LIN {X 0,Y 362.769,Z 567.893,A -85,B 0,C 180,E1 -12881.17,E2 -12881.17} C_VEL
LIN {X 0,Y 361.723,Z 575.209,A -85,B 0,C 180,E1 -12883.722,E2 -12883.722} C_VEL
LIN {X 0,Y 361.091,Z 580.078,A -85,B 0,C 180,E1 -12885.812,E2 -12885.812} C_VEL
LIN {X 0,Y 360.592,Z 584.335,A -85,B 0,C 180,E1 -12888.17,E2 -12888.17} C_VEL
LIN {X 0,Y 360.281,Z 587.529,A -85,B 0,C 180,E1 -12890.556,E2 -12890.556} C_VEL
LIN {X 0,Y 360.062,Z 589.612,A -85,B 0,C 180,E1 -12892.977,E2 -12892.977} C_VEL
LIN {X 0,Y 360.017,Z 590.544,A -85,B 0,C 180,E1 -12895.433,E2 -12895.433} C_VEL
LIN {X 0,Y 360.084,Z 590.365,A -85,B 0,C 180,E1 -12897.931,E2 -12897.931} C_VEL
LIN {X 0,Y 360.211,Z 588.944,A -85,B 0,C 180,E1 -12900.482,E2 -12900.482} C_VEL
LIN {X 0,Y 360.536,Z 586.171,A -85,B 0,C 180,E1 -12903.079,E2 -12903.079} C_VEL
LIN {X 0,Y 361.081,Z 581.98,A -85,B 0,C 180,E1 -12905.725,E2 -12905.725} C_VEL
LIN {X 0,Y 361.82,Z 576.187,A -85,B 0,C 180,E1 -12908.43,E2 -12908.43} C_VEL
LIN {X 0,Y 362.912,Z 569.264,A -85,B 0,C 180,E1 -12910.952,E2 -12910.952} C_VEL
LIN {X 0,Y 364.311,Z 561.304,A -85,B 0,C 180,E1 -12913.307,E2 -12913.307} C_VEL
LIN {X 0,Y 366.113,Z 551.646,A -85,B 0,C 180,E1 -12915.647,E2 -12915.647} C_VEL
LIN {X 0,Y 368.136,Z 541.41,A -85,B 0,C 180,E1 -12917.71,E2 -12917.71} C_VEL
LIN {X 0,Y 370.476,Z 529.462,A -85,B 0,C 180,E1 -12919.738,E2 -12919.738} C_VEL
LIN {X 0,Y 372.823,Z 516.873,A -85,B 0,C 180,E1 -12921.532,E2 -12921.532} C_VEL
LIN {X 0,Y 375.168,Z 504.129,A -85,B 0,C 180,E1 -12923.058,E2 -12923.058} C_VEL
LIN {X 0,Y 377.529,Z 489.396,A -85,B 0,C 180,E1 -12924.53,E2 -12924.53} C_VEL
LIN {X 0,Y 379.798,Z 473.918,A -85,B 0,C 180,E1 -12925.782,E2 -12925.782} C_VEL
LIN {X 0,Y 381.548,Z 459.656,A -85,B 0,C 180,E1 -12926.719,E2 -12926.719} C_VEL
LIN {X 0,Y 383.185,Z 443.468,A -85,B 0,C 180,E1 -12927.561,E2 -12927.561} C_VEL
LIN {X 0,Y 384.533,Z 426.825,A -85,B 0,C 180,E1 -12928.196,E2 -12928.196} C_VEL
LIN {X 0,Y 385.454,Z 409.688,A -85,B 0,C 180,E1 -12928.632,E2 -12928.632} C_VEL
LIN {X 0,Y 390.375,Z 262.96,A -85,B 0,C 180,E1 -12931.532,E2 -12931.532} C_VEL
LIN {X 0,Y 381.789,Z 246.096,A -85,B 0,C 180,E1 -12932.964,E2 -12932.964} C_VEL
LIN {X 0,Y 375.213,Z 234.438,A -85,B 0,C 180,E1 -12934.104,E2 -12934.104} C_VEL
LIN {X 0,Y 367.237,Z 221.553,A -85,B 0,C 180,E1 -12935.553,E2 -12935.553} C_VEL
LIN {X 0,Y 365.03,Z 218.312,A -85,B 0,C 180,E1 -12935.963,E2 -12935.963} C_VEL
LIN {X 0,Y 362.546,Z 214.885,A -85,B 0,C 180,E1 -12936.433,E2 -12936.433} C_VEL
LIN {X 0,Y 362.042,Z 213.576,A -85,B 0,C 180,E1 -12936.55,E2 -12936.55} C_VEL
LIN {X 0,Y 361.879,Z 212.722,A -85,B 0,C 180,E1 -12936.766,E2 -12936.766} C_VEL
LIN {X 0,Y 361.879,Z 212.713,A -85,B 0,C 180,E1 -12940.722,E2 -12940.722} C_VEL
LIN {X 0,Y 361.937,Z 212.702,A -85,B 0,C 180,E1 -12944.226,E2 -12944.226} C_VEL
LIN {X 0,Y 361.993,Z 212.706,A -85,B 0,C 180,E1 -12946.528,E2 -12946.528} C_VEL
LIN {X 0,Y 361.994,Z 212.706,A -85,B 0,C 180,E1 -12949.937,E2 -12949.937} C_VEL
LIN {X 0,Y 362.142,Z 212.683,A -85,B 0,C 180,E1 -12953.313,E2 -12953.313} C_VEL
LIN {X 0,Y 362.274,Z 212.669,A -85,B 0,C 180,E1 -12957.776,E2 -12957.776} C_VEL
LIN {X 0,Y 362.421,Z 212.652,A -85,B 0,C 180,E1 -12960,E2 -12960} C_VEL
LIN {X 0,Y 362.274,Z 212.671,A -85,B 0,C 180,E1 -12962.224,E2 -12962.224} C_VEL
LIN {X 0,Y 362.157,Z 212.687,A -85,B 0,C 180,E1 -12966.686,E2 -12966.686} C_VEL
LIN {X 0,Y 362.025,Z 212.703,A -85,B 0,C 180,E1 -12970.062,E2 -12970.062} C_VEL
LIN {X 0,Y 361.992,Z 212.703,A -85,B 0,C 180,E1 -12973.899,E2 -12973.899} C_VEL
LIN {X 0,Y 361.962,Z 212.711,A -85,B 0,C 180,E1 -12977.939,E2 -12977.939} C_VEL
LIN {X 0,Y 361.886,Z 212.717,A -85,B 0,C 180,E1 -12981.653,E2 -12981.653} C_VEL
LIN {X 0,Y 361.923,Z 212.715,A -85,B 0,C 180,E1 -12985.29,E2 -12985.29} C_VEL
LIN {X 0,Y 361.903,Z 212.721,A -85,B 0,C 180,E1 -12987.779,E2 -12987.779} C_VEL
LIN {X 0,Y 361.832,Z 212.726,A -85,B 0,C 180,E1 -12991.63,E2 -12991.63} C_VEL
LIN {X 0,Y 361.869,Z 212.725,A -85,B 0,C 180,E1 -12995.345,E2 -12995.345} C_VEL
LIN {X 0,Y 361.865,Z 212.73,A -85,B 0,C 180,E1 -12999.027,E2 -12999.027} C_VEL
LIN {X 0,Y 361.831,Z 212.734,A -85,B 0,C 180,E1 -13002.829,E2 -13002.829} C_VEL
LIN {X 0,Y 361.843,Z 212.773,A -85,B 0,C 180,E1 -13006.82,E2 -13006.82} C_VEL
LIN {X 0,Y 367.527,Z 227.558,A -85,B 0,C 180,E1 -13010.269,E2 -13010.269} C_VEL
LIN {X 0,Y 376.278,Z 242.828,A -85,B 0,C 180,E1 -13011.891,E2 -13011.891} C_VEL
LIN {X 0,Y 384.124,Z 257.902,A -85,B 0,C 180,E1 -13013.252,E2 -13013.252} C_VEL
LIN {X 0,Y 389.455,Z 269.218,A -85,B 0,C 180,E1 -13014.151,E2 -13014.151} C_VEL
LIN {X 0,Y 390.123,Z 274.919,A -85,B 0,C 180,E1 -13014.361,E2 -13014.361} C_VEL
LIN {X 0,Y 384.621,Z 436.732,A -85,B 0,C 180,E1 -13017.579,E2 -13017.579} C_VEL
LIN {X 0,Y 383.351,Z 452.919,A -85,B 0,C 180,E1 -13018.077,E2 -13018.077} C_VEL
LIN {X 0,Y 381.853,Z 468.395,A -85,B 0,C 180,E1 -13018.75,E2 -13018.75} C_VEL
LIN {X 0,Y 380.022,Z 483.398,A -85,B 0,C 180,E1 -13019.586,E2 -13019.586} C_VEL
LIN {X 0,Y 377.904,Z 498.273,A -85,B 0,C 180,E1 -13020.627,E2 -13020.627} C_VEL
LIN {X 0,Y 375.599,Z 513.155,A -85,B 0,C 180,E1 -13021.923,E2 -13021.923} C_VEL
LIN {X 0,Y 373.038,Z 527.462,A -85,B 0,C 180,E1 -13023.421,E2 -13023.421} C_VEL
LIN {X 0,Y 370.694,Z 540.406,A -85,B 0,C 180,E1 -13025.05,E2 -13025.05} C_VEL
LIN {X 0,Y 368.649,Z 551.565,A -85,B 0,C 180,E1 -13026.698,E2 -13026.698} C_VEL
LIN {X 0,Y 366.587,Z 562.673,A -85,B 0,C 180,E1 -13028.639,E2 -13028.639} C_VEL
LIN {X 0,Y 364.623,Z 573.214,A -85,B 0,C 180,E1 -13030.814,E2 -13030.814} C_VEL
LIN {X 0,Y 363.105,Z 582.549,A -85,B 0,C 180,E1 -13033.123,E2 -13033.123} C_VEL
LIN {X 0,Y 361.954,Z 590.186,A -85,B 0,C 180,E1 -13035.38,E2 -13035.38} C_VEL
LIN {X 0,Y 361.04,Z 597.839,A -85,B 0,C 180,E1 -13038.207,E2 -13038.207} C_VEL
LIN {X 0,Y 360.52,Z 603.683,A -85,B 0,C 180,E1 -13041.028,E2 -13041.028} C_VEL
LIN {X 0,Y 360.379,Z 607.096,A -85,B 0,C 180,E1 -13043.281,E2 -13043.281} C_VEL
LIN {X 0,Y 360.298,Z 609.553,A -85,B 0,C 180,E1 -13045.525,E2 -13045.525} C_VEL
LIN {X 0,Y 360.27,Z 610.947,A -85,B 0,C 180,E1 -13047.764,E2 -13047.764} C_VEL
LIN {X 0,Y 360.356,Z 611.428,A -85,B 0,C 180,E1 -13050,E2 -13050} C_VEL
LIN {X 0,Y 360.272,Z 610.861,A -85,B 0,C 180,E1 -13052.236,E2 -13052.236} C_VEL
LIN {X 0,Y 360.298,Z 609.372,A -85,B 0,C 180,E1 -13054.475,E2 -13054.475} C_VEL
LIN {X 0,Y 360.379,Z 606.819,A -85,B 0,C 180,E1 -13056.72,E2 -13056.72} C_VEL
LIN {X 0,Y 360.521,Z 603.263,A -85,B 0,C 180,E1 -13058.972,E2 -13058.972} C_VEL
LIN {X 0,Y 360.875,Z 598.584,A -85,B 0,C 180,E1 -13061.23,E2 -13061.23} C_VEL
LIN {X 0,Y 361.623,Z 592.232,A -85,B 0,C 180,E1 -13063.657,E2 -13063.657} C_VEL
LIN {X 0,Y 362.564,Z 584.596,A -85,B 0,C 180,E1 -13066.035,E2 -13066.035} C_VEL
LIN {X 0,Y 363.903,Z 575.912,A -85,B 0,C 180,E1 -13068.277,E2 -13068.277} C_VEL
LIN {X 0,Y 365.602,Z 565.37,A -85,B 0,C 180,E1 -13070.538,E2 -13070.538} C_VEL
LIN {X 0,Y 367.5,Z 554.478,A -85,B 0,C 180,E1 -13072.487,E2 -13072.487} C_VEL
LIN {X 0,Y 369.418,Z 543.389,A -85,B 0,C 180,E1 -13074.185,E2 -13074.185} C_VEL
LIN {X 0,Y 371.553,Z 531.128,A -85,B 0,C 180,E1 -13075.788,E2 -13075.788} C_VEL
LIN {X 0,Y 373.767,Z 517.501,A -85,B 0,C 180,E1 -13077.279,E2 -13077.279} C_VEL
LIN {X 0,Y 375.967,Z 503.055,A -85,B 0,C 180,E1 -13078.591,E2 -13078.591} C_VEL
LIN {X 0,Y 377.997,Z 488.557,A -85,B 0,C 180,E1 -13079.672,E2 -13079.672} C_VEL
LIN {X 0,Y 379.777,Z 473.42,A -85,B 0,C 180,E1 -13080.591,E2 -13080.591} C_VEL
LIN {X 0,Y 381.381,Z 455.748,A -85,B 0,C 180,E1 -13081.41,E2 -13081.41} C_VEL
LIN {X 0,Y 382.692,Z 438.69,A -85,B 0,C 180,E1 -13081.947,E2 -13081.947} C_VEL
LIN {X 0,Y 383.543,Z 416.513,A -85,B 0,C 180,E1 -13082.407,E2 -13082.407} C_VEL
LIN {X 0,Y 387.858,Z 273.203,A -85,B 0,C 180,E1 -13085.197,E2 -13085.197} C_VEL
LIN {X 0,Y 386.788,Z 267.489,A -85,B 0,C 180,E1 -13085.431,E2 -13085.431} C_VEL
LIN {X 0,Y 376.132,Z 245.181,A -85,B 0,C 180,E1 -13087.042,E2 -13087.042} C_VEL
LIN {X 0,Y 367.589,Z 229.114,A -85,B 0,C 180,E1 -13088.383,E2 -13088.383} C_VEL
LIN {X 0,Y 362.976,Z 216.179,A -85,B 0,C 180,E1 -13090.964,E2 -13090.964} C_VEL
LIN {X 0,Y 361.842,Z 212.725,A -85,B 0,C 180,E1 -13091.692,E2 -13091.692} C_VEL
LIN {X 0,Y 361.814,Z 212.718,A -85,B 0,C 180,E1 -13095.631,E2 -13095.631} C_VEL
LIN {X 0,Y 361.827,Z 212.716,A -85,B 0,C 180,E1 -13099.246,E2 -13099.246} C_VEL
LIN {X 0,Y 361.863,Z 212.71,A -85,B 0,C 180,E1 -13102.982,E2 -13102.982} C_VEL
LIN {X 0,Y 361.856,Z 212.721,A -85,B 0,C 180,E1 -13106.631,E2 -13106.631} C_VEL
LIN {X 0,Y 361.871,Z 212.714,A -85,B 0,C 180,E1 -13109.672,E2 -13109.672} C_VEL
LIN {X 0,Y 361.951,Z 212.692,A -85,B 0,C 180,E1 -13113.475,E2 -13113.475} C_VEL
LIN {X 0,Y 361.888,Z 212.721,A -85,B 0,C 180,E1 -13117.145,E2 -13117.145} C_VEL
LIN {X 0,Y 361.883,Z 212.693,A -85,B 0,C 180,E1 -13120.722,E2 -13120.722} C_VEL
LIN {X 0,Y 361.941,Z 212.713,A -85,B 0,C 180,E1 -13124.226,E2 -13124.226} C_VEL
LIN {X 0,Y 361.996,Z 212.689,A -85,B 0,C 180,E1 -13126.528,E2 -13126.528} C_VEL
LIN {X 0,Y 361.997,Z 212.686,A -85,B 0,C 180,E1 -13129.937,E2 -13129.937} C_VEL
LIN {X 0,Y 362.146,Z 212.684,A -85,B 0,C 180,E1 -13133.313,E2 -13133.313} C_VEL
LIN {X 0,Y 362.277,Z 212.634,A -85,B 0,C 180,E1 -13137.776,E2 -13137.776} C_VEL
LIN {X 0,Y 362.423,Z 212.643,A -85,B 0,C 180,E1 -13140,E2 -13140} C_VEL
LIN {X 0,Y 362.277,Z 212.671,A -85,B 0,C 180,E1 -13142.224,E2 -13142.224} C_VEL
LIN {X 0,Y 362.16,Z 212.678,A -85,B 0,C 180,E1 -13146.686,E2 -13146.686} C_VEL
LIN {X 0,Y 362.028,Z 212.694,A -85,B 0,C 180,E1 -13150.062,E2 -13150.062} C_VEL
LIN {X 0,Y 361.996,Z 212.697,A -85,B 0,C 180,E1 -13153.899,E2 -13153.899} C_VEL
LIN {X 0,Y 361.965,Z 212.691,A -85,B 0,C 180,E1 -13157.939,E2 -13157.939} C_VEL
LIN {X 0,Y 361.89,Z 212.717,A -85,B 0,C 180,E1 -13161.653,E2 -13161.653} C_VEL
LIN {X 0,Y 361.926,Z 212.696,A -85,B 0,C 180,E1 -13165.29,E2 -13165.29} C_VEL
LIN {X 0,Y 361.921,Z 212.712,A -85,B 0,C 180,E1 -13167.778,E2 -13167.778} C_VEL
LIN {X 0,Y 361.845,Z 212.711,A -85,B 0,C 180,E1 -13171.285,E2 -13171.285} C_VEL
LIN {X 0,Y 361.853,Z 212.723,A -85,B 0,C 180,E1 -13174.28,E2 -13174.28} C_VEL
LIN {X 0,Y 361.863,Z 212.712,A -85,B 0,C 180,E1 -13177.223,E2 -13177.223} C_VEL
LIN {X 0,Y 361.835,Z 212.724,A -85,B 0,C 180,E1 -13180.756,E2 -13180.756} C_VEL
LIN {X 0,Y 361.815,Z 212.717,A -85,B 0,C 180,E1 -13184.369,E2 -13184.369} C_VEL
LIN {X 0,Y 361.834,Z 212.721,A -85,B 0,C 180,E1 -13187.568,E2 -13187.568} C_VEL
LIN {X 0,Y 361.867,Z 212.72,A -85,B 0,C 180,E1 -13190.974,E2 -13190.974} C_VEL
LIN {X 0,Y 361.873,Z 212.71,A -85,B 0,C 180,E1 -13194.655,E2 -13194.655} C_VEL
LIN {X 0,Y 361.836,Z 212.714,A -85,B 0,C 180,E1 -13198.371,E2 -13198.371} C_VEL
LIN {X 0,Y 361.9,Z 212.721,A -85,B 0,C 180,E1 -13200.955,E2 -13200.955} C_VEL
LIN {X 0,Y 361.953,Z 212.705,A -85,B 0,C 180,E1 -13203.475,E2 -13203.475} C_VEL
LIN {X 0,Y 361.892,Z 212.714,A -85,B 0,C 180,E1 -13207.145,E2 -13207.145} C_VEL
LIN {X 0,Y 361.887,Z 212.689,A -85,B 0,C 180,E1 -13210.722,E2 -13210.722} C_VEL
LIN {X 0,Y 361.933,Z 212.711,A -85,B 0,C 180,E1 -13213.066,E2 -13213.066} C_VEL
LIN {X 0,Y 362.024,Z 212.683,A -85,B 0,C 180,E1 -13217.039,E2 -13217.039} C_VEL
LIN {X 0,Y 363.054,Z 215.611,A -85,B 0,C 180,E1 -13217.248,E2 -13217.248} C_VEL
LIN {X 0,Y 364.548,Z 217.745,A -85,B 0,C 180,E1 -13217.479,E2 -13217.479} C_VEL
LIN {X 0,Y 373.522,Z 232.837,A -85,B 0,C 180,E1 -13218.87,E2 -13218.87} C_VEL
LIN {X 0,Y 381.962,Z 248.896,A -85,B 0,C 180,E1 -13220.142,E2 -13220.142} C_VEL
LIN {X 0,Y 388.027,Z 261.925,A -85,B 0,C 180,E1 -13221.052,E2 -13221.052} C_VEL
LIN {X 0,Y 383.18,Z 416.866,A -85,B 0,C 180,E1 -13224.078,E2 -13224.078} C_VEL
LIN {X 0,Y 382.141,Z 433.477,A -85,B 0,C 180,E1 -13224.591,E2 -13224.591} C_VEL
LIN {X 0,Y 380.8,Z 449.353,A -85,B 0,C 180,E1 -13225.284,E2 -13225.284} C_VEL
LIN {X 0,Y 379.228,Z 464.561,A -85,B 0,C 180,E1 -13226.148,E2 -13226.148} C_VEL
LIN {X 0,Y 377.475,Z 479.265,A -85,B 0,C 180,E1 -13227.198,E2 -13227.198} C_VEL
LIN {X 0,Y 375.491,Z 493,A -85,B 0,C 180,E1 -13228.391,E2 -13228.391} C_VEL
LIN {X 0,Y 373.256,Z 507.153,A -85,B 0,C 180,E1 -13229.865,E2 -13229.865} C_VEL
LIN {X 0,Y 371.296,Z 519.204,A -85,B 0,C 180,E1 -13231.355,E2 -13231.355} C_VEL
LIN {X 0,Y 368.932,Z 532.288,A -85,B 0,C 180,E1 -13233.276,E2 -13233.276} C_VEL
LIN {X 0,Y 366.965,Z 543.218,A -85,B 0,C 180,E1 -13235.201,E2 -13235.201} C_VEL
LIN {X 0,Y 365.295,Z 552.773,A -85,B 0,C 180,E1 -13237.184,E2 -13237.184} C_VEL
LIN {X 0,Y 364.07,Z 559.988,A -85,B 0,C 180,E1 -13238.919,E2 -13238.919} C_VEL
LIN {X 0,Y 362.924,Z 563.011,A -85,B 0,C 180,E1 -13239.699,E2 -13239.699} C_VEL
LIN {X 0,Y 356.43,Z 571.259,A -85,B 0,C 180,E1 -13242.006,E2 -13242.006} C_VEL
LIN {X 0,Y 355.052,Z 573.747,A -85,B 0,C 180,E1 -13242.844,E2 -13242.844} C_VEL
LIN {X 0,Y 354.865,Z 574.488,A -85,B 0,C 180,E1 -13243.134,E2 -13243.134} C_VEL
LIN {X 0,Y 354.076,Z 580.085,A -85,B 0,C 180,E1 -13245.542,E2 -13245.542} C_VEL
LIN {X 0,Y 353.644,Z 583.644,A -85,B 0,C 180,E1 -13247.464,E2 -13247.464} C_VEL
LIN {X 0,Y 353.257,Z 586.927,A -85,B 0,C 180,E1 -13249.767,E2 -13249.767} C_VEL
LIN {X 0,Y 352.994,Z 589.314,A -85,B 0,C 180,E1 -13252.227,E2 -13252.227} C_VEL
LIN {X 0,Y 352.916,Z 590.638,A -85,B 0,C 180,E1 -13254.72,E2 -13254.72} C_VEL
LIN {X 0,Y 352.949,Z 590.735,A -85,B 0,C 180,E1 -13257.256,E2 -13257.256} C_VEL
LIN {X 0,Y 353.05,Z 589.663,A -85,B 0,C 180,E1 -13259.845,E2 -13259.845} C_VEL
LIN {X 0,Y 353.334,Z 587.334,A -85,B 0,C 180,E1 -13262.482,E2 -13262.482} C_VEL
LIN {X 0,Y 353.885,Z 583.591,A -85,B 0,C 180,E1 -13265.164,E2 -13265.164} C_VEL
LIN {X 0,Y 354.582,Z 578.249,A -85,B 0,C 180,E1 -13267.91,E2 -13267.91} C_VEL
LIN {X 0,Y 355.418,Z 572.986,A -85,B 0,C 180,E1 -13270.04,E2 -13270.04} C_VEL
LIN {X 0,Y 356.46,Z 566.926,A -85,B 0,C 180,E1 -13272.093,E2 -13272.093} C_VEL
LIN {X 0,Y 358.153,Z 558.136,A -85,B 0,C 180,E1 -13274.548,E2 -13274.548} C_VEL
LIN {X 0,Y 359.902,Z 549.284,A -85,B 0,C 180,E1 -13276.618,E2 -13276.618} C_VEL
LIN {X 0,Y 362.163,Z 538.628,A -85,B 0,C 180,E1 -13278.716,E2 -13278.716} C_VEL
LIN {X 0,Y 364.59,Z 526.833,A -85,B 0,C 180,E1 -13280.665,E2 -13280.665} C_VEL
LIN {X 0,Y 366.84,Z 514.974,A -85,B 0,C 180,E1 -13282.316,E2 -13282.316} C_VEL
LIN {X 0,Y 369.3,Z 501.917,A -85,B 0,C 180,E1 -13283.847,E2 -13283.847} C_VEL
LIN {X 0,Y 371.611,Z 488.087,A -85,B 0,C 180,E1 -13285.213,E2 -13285.213} C_VEL
LIN {X 0,Y 373.844,Z 473.322,A -85,B 0,C 180,E1 -13286.411,E2 -13286.411} C_VEL
LIN {X 0,Y 375.816,Z 457.752,A -85,B 0,C 180,E1 -13287.424,E2 -13287.424} C_VEL
LIN {X 0,Y 377.404,Z 441.921,A -85,B 0,C 180,E1 -13288.233,E2 -13288.233} C_VEL
LIN {X 0,Y 378.794,Z 425.309,A -85,B 0,C 180,E1 -13288.845,E2 -13288.845} C_VEL
LIN {X 0,Y 379.651,Z 408.154,A -85,B 0,C 180,E1 -13289.274,E2 -13289.274} C_VEL
LIN {X 0,Y 384.65,Z 265.3,A -85,B 0,C 180,E1 -13292.141,E2 -13292.141} C_VEL
LIN {X 0,Y 377.068,Z 250.316,A -85,B 0,C 180,E1 -13293.451,E2 -13293.451} C_VEL
LIN {X 0,Y 369.948,Z 237.666,A -85,B 0,C 180,E1 -13294.733,E2 -13294.733} C_VEL
LIN {X 0,Y 363.101,Z 226.601,A -85,B 0,C 180,E1 -13296.017,E2 -13296.017} C_VEL
LIN {X 0,Y 359.879,Z 221.971,A -85,B 0,C 180,E1 -13296.639,E2 -13296.639} C_VEL
LIN {X 0,Y 357.501,Z 218.319,A -85,B 0,C 180,E1 -13297.116,E2 -13297.116} C_VEL
LIN {X 0,Y 355.465,Z 215.85,A -85,B 0,C 180,E1 -13297.515,E2 -13297.515} C_VEL
LIN {X 0,Y 354.797,Z 213.63,A -85,B 0,C 180,E1 -13297.738,E2 -13297.738} C_VEL
LIN {X 0,Y 354.841,Z 213.591,A -85,B 0,C 180,E1 -13301.525,E2 -13301.525} C_VEL
LIN {X 0,Y 354.913,Z 213.58,A -85,B 0,C 180,E1 -13305.083,E2 -13305.083} C_VEL
LIN {X 0,Y 354.927,Z 213.573,A -85,B 0,C 180,E1 -13308.579,E2 -13308.579} C_VEL
LIN {X 0,Y 355.055,Z 213.57,A -85,B 0,C 180,E1 -13312.036,E2 -13312.036} C_VEL
LIN {X 0,Y 355.077,Z 213.568,A -85,B 0,C 180,E1 -13314.32,E2 -13314.32} C_VEL
LIN {X 0,Y 355.237,Z 213.546,A -85,B 0,C 180,E1 -13317.732,E2 -13317.732} C_VEL
LIN {X 0,Y 355.391,Z 213.528,A -85,B 0,C 180,E1 -13320,E2 -13320} C_VEL
LIN {X 0,Y 355.237,Z 213.547,A -85,B 0,C 180,E1 -13322.268,E2 -13322.268} C_VEL
LIN {X 0,Y 355.12,Z 213.563,A -85,B 0,C 180,E1 -13326.82,E2 -13326.82} C_VEL
LIN {X 0,Y 354.972,Z 213.579,A -85,B 0,C 180,E1 -13330.264,E2 -13330.264} C_VEL
LIN {X 0,Y 354.937,Z 213.582,A -85,B 0,C 180,E1 -13334.019,E2 -13334.019} C_VEL
LIN {X 0,Y 354.917,Z 213.587,A -85,B 0,C 180,E1 -13338.109,E2 -13338.109} C_VEL
LIN {X 0,Y 354.829,Z 213.596,A -85,B 0,C 180,E1 -13342.106,E2 -13342.106} C_VEL
LIN {X 0,Y 354.894,Z 213.59,A -85,B 0,C 180,E1 -13345.828,E2 -13345.828} C_VEL
LIN {X 0,Y 354.812,Z 213.6,A -85,B 0,C 180,E1 -13349.682,E2 -13349.682} C_VEL
LIN {X 0,Y 354.801,Z 213.603,A -85,B 0,C 180,E1 -13353.702,E2 -13353.702} C_VEL
LIN {X 0,Y 354.793,Z 213.607,A -85,B 0,C 180,E1 -13356.46,E2 -13356.46} C_VEL
LIN {X 0,Y 354.819,Z 213.606,A -85,B 0,C 180,E1 -13359.424,E2 -13359.424} C_VEL
LIN {X 0,Y 354.783,Z 213.613,A -85,B 0,C 180,E1 -13362.868,E2 -13362.868} C_VEL
LIN {X 0,Y 354.792,Z 213.641,A -85,B 0,C 180,E1 -13365.814,E2 -13365.814} C_VEL
LIN {X 0,Y 360.125,Z 227.357,A -85,B 0,C 180,E1 -13369.185,E2 -13369.185} C_VEL
LIN {X 0,Y 367.513,Z 239.811,A -85,B 0,C 180,E1 -13370.623,E2 -13370.623} C_VEL
LIN {X 0,Y 375.875,Z 255.03,A -85,B 0,C 180,E1 -13372.154,E2 -13372.154} C_VEL
LIN {X 0,Y 384.139,Z 272.385,A -85,B 0,C 180,E1 -13373.61,E2 -13373.61} C_VEL
LIN {X 0,Y 384.462,Z 276.603,A -85,B 0,C 180,E1 -13373.751,E2 -13373.751} C_VEL
LIN {X 0,Y 378.761,Z 436.245,A -85,B 0,C 180,E1 -13376.966,E2 -13376.966} C_VEL
LIN {X 0,Y 377.442,Z 452.666,A -85,B 0,C 180,E1 -13377.477,E2 -13377.477} C_VEL
LIN {X 0,Y 375.956,Z 467.472,A -85,B 0,C 180,E1 -13378.124,E2 -13378.124} C_VEL
LIN {X 0,Y 374.219,Z 481.6,A -85,B 0,C 180,E1 -13378.906,E2 -13378.906} C_VEL
LIN {X 0,Y 371.996,Z 496.641,A -85,B 0,C 180,E1 -13379.957,E2 -13379.957} C_VEL
LIN {X 0,Y 369.786,Z 510.587,A -85,B 0,C 180,E1 -13381.155,E2 -13381.155} C_VEL
LIN {X 0,Y 367.362,Z 523.948,A -85,B 0,C 180,E1 -13382.515,E2 -13382.515} C_VEL
LIN {X 0,Y 364.801,Z 537.406,A -85,B 0,C 180,E1 -13384.16,E2 -13384.16} C_VEL
LIN {X 0,Y 362.4,Z 549.736,A -85,B 0,C 180,E1 -13385.968,E2 -13385.968} C_VEL
LIN {X 0,Y 360.152,Z 561.093,A -85,B 0,C 180,E1 -13387.937,E2 -13387.937} C_VEL
LIN {X 0,Y 358.026,Z 572.104,A -85,B 0,C 180,E1 -13390.208,E2 -13390.208} C_VEL
LIN {X 0,Y 356.435,Z 581.396,A -85,B 0,C 180,E1 -13392.501,E2 -13392.501} C_VEL
LIN {X 0,Y 354.994,Z 590.041,A -85,B 0,C 180,E1 -13395.087,E2 -13395.087} C_VEL
LIN {X 0,Y 354.162,Z 596.272,A -85,B 0,C 180,E1 -13397.392,E2 -13397.392} C_VEL
LIN {X 0,Y 353.567,Z 601.354,A -85,B 0,C 180,E1 -13399.695,E2 -13399.695} C_VEL
LIN {X 0,Y 353.358,Z 605.344,A -85,B 0,C 180,E1 -13401.997,E2 -13401.997} C_VEL
LIN {X 0,Y 353.239,Z 608.251,A -85,B 0,C 180,E1 -13404.291,E2 -13404.291} C_VEL
LIN {X 0,Y 353.191,Z 610.189,A -85,B 0,C 180,E1 -13406.578,E2 -13406.578} C_VEL
LIN {X 0,Y 353.218,Z 611.093,A -85,B 0,C 180,E1 -13408.86,E2 -13408.86} C_VEL
LIN {X 0,Y 353.219,Z 611.068,A -85,B 0,C 180,E1 -13411.14,E2 -13411.14} C_VEL
LIN {X 0,Y 353.191,Z 610.008,A -85,B 0,C 180,E1 -13413.423,E2 -13413.423} C_VEL
LIN {X 0,Y 353.275,Z 607.799,A -85,B 0,C 180,E1 -13415.908,E2 -13415.908} C_VEL
LIN {X 0,Y 353.359,Z 604.923,A -85,B 0,C 180,E1 -13418.003,E2 -13418.003} C_VEL
LIN {X 0,Y 353.556,Z 600.84,A -85,B 0,C 180,E1 -13420.306,E2 -13420.306} C_VEL
LIN {X 0,Y 354.369,Z 594.074,A -85,B 0,C 180,E1 -13423.184,E2 -13423.184} C_VEL
LIN {X 0,Y 355.196,Z 587.202,A -85,B 0,C 180,E1 -13425.493,E2 -13425.493} C_VEL
LIN {X 0,Y 356.527,Z 578.965,A -85,B 0,C 180,E1 -13427.791,E2 -13427.791} C_VEL
LIN {X 0,Y 357.876,Z 570.499,A -85,B 0,C 180,E1 -13429.801,E2 -13429.801} C_VEL
LIN {X 0,Y 359.666,Z 560.51,A -85,B 0,C 180,E1 -13431.794,E2 -13431.794} C_VEL
LIN {X 0,Y 361.831,Z 548.841,A -85,B 0,C 180,E1 -13433.768,E2 -13433.768} C_VEL
LIN {X 0,Y 364.076,Z 536.102,A -85,B 0,C 180,E1 -13435.589,E2 -13435.589} C_VEL
LIN {X 0,Y 366.299,Z 523.51,A -85,B 0,C 180,E1 -13437.109,E2 -13437.109} C_VEL
LIN {X 0,Y 368.698,Z 508.886,A -85,B 0,C 180,E1 -13438.57,E2 -13438.57} C_VEL
LIN {X 0,Y 371.003,Z 493.57,A -85,B 0,C 180,E1 -13439.819,E2 -13439.819} C_VEL
LIN {X 0,Y 372.966,Z 478.411,A -85,B 0,C 180,E1 -13440.818,E2 -13440.818} C_VEL
LIN {X 0,Y 374.63,Z 462.494,A -85,B 0,C 180,E1 -13441.647,E2 -13441.647} C_VEL
LIN {X 0,Y 375.968,Z 447.412,A -85,B 0,C 180,E1 -13442.231,E2 -13442.231} C_VEL
LIN {X 0,Y 377.001,Z 431.543,A -85,B 0,C 180,E1 -13442.646,E2 -13442.646} C_VEL
LIN {X 0,Y 381.929,Z 274.277,A -85,B 0,C 180,E1 -13445.762,E2 -13445.762} C_VEL
LIN {X 0,Y 380.971,Z 269.911,A -85,B 0,C 180,E1 -13445.959,E2 -13445.959} C_VEL
LIN {X 0,Y 370.041,Z 247.21,A -85,B 0,C 180,E1 -13447.657,E2 -13447.657} C_VEL
LIN {X 0,Y 360.223,Z 228.821,A -85,B 0,C 180,E1 -13449.258,E2 -13449.258} C_VEL
LIN {X 0,Y 354.812,Z 213.593,A -85,B 0,C 180,E1 -13452.433,E2 -13452.433} C_VEL
LIN {X 0,Y 354.764,Z 213.596,A -85,B 0,C 180,E1 -13456.103,E2 -13456.103} C_VEL
LIN {X 0,Y 354.779,Z 213.594,A -85,B 0,C 180,E1 -13459.178,E2 -13459.178} C_VEL
LIN {X 0,Y 354.799,Z 213.597,A -85,B 0,C 180,E1 -13462.404,E2 -13462.404} C_VEL
LIN {X 0,Y 354.81,Z 213.595,A -85,B 0,C 180,E1 -13464.941,E2 -13464.941} C_VEL
LIN {X 0,Y 354.791,Z 213.585,A -85,B 0,C 180,E1 -13468.405,E2 -13468.405} C_VEL
LIN {X 0,Y 354.844,Z 213.596,A -85,B 0,C 180,E1 -13471.619,E2 -13471.619} C_VEL
LIN {X 0,Y 354.897,Z 213.567,A -85,B 0,C 180,E1 -13474.173,E2 -13474.173} C_VEL
LIN {X 0,Y 354.832,Z 213.598,A -85,B 0,C 180,E1 -13477.894,E2 -13477.894} C_VEL
LIN {X 0,Y 354.887,Z 213.573,A -85,B 0,C 180,E1 -13481.908,E2 -13481.908} C_VEL
LIN {X 0,Y 354.941,Z 213.576,A -85,B 0,C 180,E1 -13485.981,E2 -13485.981} C_VEL
LIN {X 0,Y 354.953,Z 213.562,A -85,B 0,C 180,E1 -13489.735,E2 -13489.735} C_VEL
LIN {X 0,Y 355.109,Z 213.561,A -85,B 0,C 180,E1 -13493.18,E2 -13493.18} C_VEL
LIN {X 0,Y 355.24,Z 213.509,A -85,B 0,C 180,E1 -13497.732,E2 -13497.732} C_VEL
LIN {X 0,Y 355.372,Z 213.521,A -85,B 0,C 180,E1 -13500,E2 -13500} C_VEL
LIN {X 0,Y 355.241,Z 213.547,A -85,B 0,C 180,E1 -13502.268,E2 -13502.268} C_VEL
LIN {X 0,Y 355.124,Z 213.556,A -85,B 0,C 180,E1 -13506.819,E2 -13506.819} C_VEL
LIN {X 0,Y 354.975,Z 213.569,A -85,B 0,C 180,E1 -13510.264,E2 -13510.264} C_VEL
LIN {X 0,Y 354.941,Z 213.577,A -85,B 0,C 180,E1 -13514.019,E2 -13514.019} C_VEL
LIN {X 0,Y 354.92,Z 213.566,A -85,B 0,C 180,E1 -13518.108,E2 -13518.108} C_VEL
LIN {X 0,Y 354.833,Z 213.599,A -85,B 0,C 180,E1 -13522.106,E2 -13522.106} C_VEL
LIN {X 0,Y 354.897,Z 213.571,A -85,B 0,C 180,E1 -13525.827,E2 -13525.827} C_VEL
LIN {X 0,Y 354.853,Z 213.594,A -85,B 0,C 180,E1 -13529.679,E2 -13529.679} C_VEL
LIN {X 0,Y 354.804,Z 213.594,A -85,B 0,C 180,E1 -13533.702,E2 -13533.702} C_VEL
LIN {X 0,Y 354.797,Z 213.597,A -85,B 0,C 180,E1 -13536.459,E2 -13536.459} C_VEL
LIN {X 0,Y 354.823,Z 213.589,A -85,B 0,C 180,E1 -13539.424,E2 -13539.424} C_VEL
LIN {X 0,Y 354.786,Z 213.596,A -85,B 0,C 180,E1 -13542.867,E2 -13542.867} C_VEL
LIN {X 0,Y 354.766,Z 213.606,A -85,B 0,C 180,E1 -13546.104,E2 -13546.104} C_VEL
LIN {X 0,Y 354.785,Z 213.591,A -85,B 0,C 180,E1 -13549.179,E2 -13549.179} C_VEL
LIN {X 0,Y 354.805,Z 213.598,A -85,B 0,C 180,E1 -13552.403,E2 -13552.403} C_VEL
LIN {X 0,Y 354.81,Z 213.591,A -85,B 0,C 180,E1 -13554.941,E2 -13554.941} C_VEL
LIN {X 0,Y 354.792,Z 213.591,A -85,B 0,C 180,E1 -13558.405,E2 -13558.405} C_VEL
LIN {X 0,Y 354.848,Z 213.592,A -85,B 0,C 180,E1 -13561.619,E2 -13561.619} C_VEL
LIN {X 0,Y 354.899,Z 213.589,A -85,B 0,C 180,E1 -13564.173,E2 -13564.173} C_VEL
LIN {X 0,Y 354.836,Z 213.599,A -85,B 0,C 180,E1 -13567.894,E2 -13567.894} C_VEL
LIN {X 0,Y 354.922,Z 213.561,A -85,B 0,C 180,E1 -13571.892,E2 -13571.892} C_VEL
LIN {X 0,Y 354.942,Z 213.559,A -85,B 0,C 180,E1 -13575.981,E2 -13575.981} C_VEL
LIN {X 0,Y 354.952,Z 213.562,A -85,B 0,C 180,E1 -13576.212,E2 -13576.212} C_VEL
LIN {X 0,Y 355.962,Z 216.419,A -85,B 0,C 180,E1 -13576.412,E2 -13576.412} C_VEL
LIN {X 0,Y 357.581,Z 218.616,A -85,B 0,C 180,E1 -13576.668,E2 -13576.668} C_VEL
LIN {X 0,Y 368.368,Z 236.593,A -85,B 0,C 180,E1 -13578.388,E2 -13578.388} C_VEL
LIN {X 0,Y 376.777,Z 252.688,A -85,B 0,C 180,E1 -13579.693,E2 -13579.693} C_VEL
LIN {X 0,Y 381.966,Z 263.819,A -85,B 0,C 180,E1 -13580.488,E2 -13580.488} C_VEL
LIN {X 0,Y 377.063,Z 417.523,A -85,B 0,C 180,E1 -13583.545,E2 -13583.545} C_VEL
LIN {X 0,Y 375.987,Z 433.957,A -85,B 0,C 180,E1 -13584.065,E2 -13584.065} C_VEL
LIN {X 0,Y 374.594,Z 449.751,A -85,B 0,C 180,E1 -13584.766,E2 -13584.766} C_VEL
LIN {X 0,Y 372.916,Z 465.402,A -85,B 0,C 180,E1 -13585.676,E2 -13585.676} C_VEL
LIN {X 0,Y 371.077,Z 480.055,A -85,B 0,C 180,E1 -13586.743,E2 -13586.743} C_VEL
LIN {X 0,Y 369.027,Z 493.685,A -85,B 0,C 180,E1 -13587.953,E2 -13587.953} C_VEL
LIN {X 0,Y 366.728,Z 507.748,A -85,B 0,C 180,E1 -13589.451,E2 -13589.451} C_VEL
LIN {X 0,Y 364.491,Z 520.723,A -85,B 0,C 180,E1 -13591.104,E2 -13591.104} C_VEL
LIN {X 0,Y 362.423,Z 531.9,A -85,B 0,C 180,E1 -13592.778,E2 -13592.778} C_VEL
LIN {X 0,Y 360.359,Z 542.836,A -85,B 0,C 180,E1 -13594.719,E2 -13594.719} C_VEL
LIN {X 0,Y 358.531,Z 552.582,A -85,B 0,C 180,E1 -13596.754,E2 -13596.754} C_VEL
LIN {X 0,Y 357.091,Z 560.823,A -85,B 0,C 180,E1 -13598.773,E2 -13598.773} C_VEL
LIN {X 0,Y 355.891,Z 567.801,A -85,B 0,C 180,E1 -13600.812,E2 -13600.812} C_VEL
LIN {X 0,Y 354.865,Z 574.488,A -85,B 0,C 180,E1 -13603.134,E2 -13603.134} C_VEL
LIN {X 0,Y 353.91,Z 576.763,A -85,B 0,C 180,E1 -13604.002,E2 -13604.002} C_VEL
LIN {X 0,Y 350.619,Z 580.187,A -85,B 0,C 180,E1 -13605.418,E2 -13605.418} C_VEL
LIN {X 0,Y 347.885,Z 582.569,A -85,B 0,C 180,E1 -13606.584,E2 -13606.584} C_VEL
LIN {X 0,Y 346.622,Z 584.136,A -85,B 0,C 180,E1 -13607.507,E2 -13607.507} C_VEL
LIN {X 0,Y 346.466,Z 584.61,A -85,B 0,C 180,E1 -13607.824,E2 -13607.824} C_VEL
LIN {X 0,Y 346.127,Z 587.751,A -85,B 0,C 180,E1 -13610.192,E2 -13610.192} C_VEL
LIN {X 0,Y 345.868,Z 589.887,A -85,B 0,C 180,E1 -13612.71,E2 -13612.71} C_VEL
LIN {X 0,Y 345.807,Z 590.926,A -85,B 0,C 180,E1 -13615.263,E2 -13615.263} C_VEL
LIN {X 0,Y 345.879,Z 590.857,A -85,B 0,C 180,E1 -13617.861,E2 -13617.861} C_VEL
LIN {X 0,Y 346.003,Z 589.494,A -85,B 0,C 180,E1 -13620.517,E2 -13620.517} C_VEL
LIN {X 0,Y 346.364,Z 586.837,A -85,B 0,C 180,E1 -13623.219,E2 -13623.219} C_VEL
LIN {X 0,Y 346.971,Z 582.766,A -85,B 0,C 180,E1 -13625.972,E2 -13625.972} C_VEL
LIN {X 0,Y 347.794,Z 577.093,A -85,B 0,C 180,E1 -13628.786,E2 -13628.786} C_VEL
LIN {X 0,Y 348.946,Z 570.708,A -85,B 0,C 180,E1 -13631.269,E2 -13631.269} C_VEL
LIN {X 0,Y 350.505,Z 562.635,A -85,B 0,C 180,E1 -13633.794,E2 -13633.794} C_VEL
LIN {X 0,Y 352.208,Z 554.461,A -85,B 0,C 180,E1 -13635.917,E2 -13635.917} C_VEL
LIN {X 0,Y 354.346,Z 544.617,A -85,B 0,C 180,E1 -13638.081,E2 -13638.081} C_VEL
LIN {X 0,Y 356.816,Z 533.188,A -85,B 0,C 180,E1 -13640.187,E2 -13640.187} C_VEL
LIN {X 0,Y 359.476,Z 520.541,A -85,B 0,C 180,E1 -13642.124,E2 -13642.124} C_VEL
LIN {X 0,Y 361.928,Z 508.343,A -85,B 0,C 180,E1 -13643.691,E2 -13643.691} C_VEL
LIN {X 0,Y 364.465,Z 494.409,A -85,B 0,C 180,E1 -13645.205,E2 -13645.205} C_VEL
LIN {X 0,Y 366.792,Z 480.447,A -85,B 0,C 180,E1 -13646.464,E2 -13646.464} C_VEL
LIN {X 0,Y 369.172,Z 463.926,A -85,B 0,C 180,E1 -13647.664,E2 -13647.664} C_VEL
LIN {X 0,Y 371.037,Z 447.731,A -85,B 0,C 180,E1 -13648.581,E2 -13648.581} C_VEL
LIN {X 0,Y 372.498,Z 431.491,A -85,B 0,C 180,E1 -13649.268,E2 -13649.268} C_VEL
LIN {X 0,Y 373.592,Z 414.816,A -85,B 0,C 180,E1 -13649.753,E2 -13649.753} C_VEL
LIN {X 0,Y 379.072,Z 267.862,A -85,B 0,C 180,E1 -13652.754,E2 -13652.754} C_VEL
LIN {X 0,Y 371.841,Z 253.524,A -85,B 0,C 180,E1 -13654.052,E2 -13654.052} C_VEL
LIN {X 0,Y 364.655,Z 240.699,A -85,B 0,C 180,E1 -13655.397,E2 -13655.397} C_VEL
LIN {X 0,Y 358.725,Z 231.244,A -85,B 0,C 180,E1 -13656.549,E2 -13656.549} C_VEL
LIN {X 0,Y 353.612,Z 223.687,A -85,B 0,C 180,E1 -13657.583,E2 -13657.583} C_VEL
LIN {X 0,Y 351.31,Z 220.512,A -85,B 0,C 180,E1 -13658.062,E2 -13658.062} C_VEL
LIN {X 0,Y 350.482,Z 219.212,A -85,B 0,C 180,E1 -13658.242,E2 -13658.242} C_VEL
LIN {X 0,Y 348.58,Z 216.958,A -85,B 0,C 180,E1 -13658.637,E2 -13658.637} C_VEL
LIN {X 0,Y 347.79,Z 214.474,A -85,B 0,C 180,E1 -13658.903,E2 -13658.903} C_VEL
LIN {X 0,Y 347.837,Z 214.472,A -85,B 0,C 180,E1 -13662.358,E2 -13662.358} C_VEL
LIN {X 0,Y 347.892,Z 214.464,A -85,B 0,C 180,E1 -13665.971,E2 -13665.971} C_VEL
LIN {X 0,Y 347.89,Z 214.461,A -85,B 0,C 180,E1 -13669.524,E2 -13669.524} C_VEL
LIN {X 0,Y 348.071,Z 214.437,A -85,B 0,C 180,E1 -13673.042,E2 -13673.042} C_VEL
LIN {X 0,Y 348.199,Z 214.422,A -85,B 0,C 180,E1 -13677.686,E2 -13677.686} C_VEL
LIN {X 0,Y 348.34,Z 214.406,A -85,B 0,C 180,E1 -13680,E2 -13680} C_VEL
LIN {X 0,Y 348.2,Z 214.423,A -85,B 0,C 180,E1 -13682.314,E2 -13682.314} C_VEL
LIN {X 0,Y 348.086,Z 214.439,A -85,B 0,C 180,E1 -13686.958,E2 -13686.958} C_VEL
LIN {X 0,Y 347.922,Z 214.455,A -85,B 0,C 180,E1 -13690.475,E2 -13690.475} C_VEL
LIN {X 0,Y 347.893,Z 214.459,A -85,B 0,C 180,E1 -13694.15,E2 -13694.15} C_VEL
LIN {X 0,Y 347.885,Z 214.461,A -85,B 0,C 180,E1 -13698.29,E2 -13698.29} C_VEL
LIN {X 0,Y 347.783,Z 214.473,A -85,B 0,C 180,E1 -13701.635,E2 -13701.635} C_VEL
LIN {X 0,Y 347.807,Z 214.472,A -85,B 0,C 180,E1 -13705.109,E2 -13705.109} C_VEL
LIN {X 0,Y 347.803,Z 214.475,A -85,B 0,C 180,E1 -13707.694,E2 -13707.694} C_VEL
LIN {X 0,Y 347.744,Z 214.483,A -85,B 0,C 180,E1 -13710.348,E2 -13710.348} C_VEL
LIN {X 0,Y 347.743,Z 214.482,A -85,B 0,C 180,E1 -13714.044,E2 -13714.044} C_VEL
LIN {X 0,Y 347.757,Z 214.485,A -85,B 0,C 180,E1 -13717.321,E2 -13717.321} C_VEL
LIN {X 0,Y 347.728,Z 214.487,A -85,B 0,C 180,E1 -13720.297,E2 -13720.297} C_VEL
LIN {X 0,Y 347.718,Z 214.491,A -85,B 0,C 180,E1 -13723.409,E2 -13723.409} C_VEL
LIN {X 0,Y 347.738,Z 214.537,A -85,B 0,C 180,E1 -13724.744,E2 -13724.744} C_VEL
LIN {X 0,Y 348.42,Z 216.79,A -85,B 0,C 180,E1 -13725.318,E2 -13725.318} C_VEL
LIN {X 0,Y 350.465,Z 221.473,A -85,B 0,C 180,E1 -13726.587,E2 -13726.587} C_VEL
LIN {X 0,Y 352.901,Z 227.382,A -85,B 0,C 180,E1 -13728.048,E2 -13728.048} C_VEL
LIN {X 0,Y 362.232,Z 242.707,A -85,B 0,C 180,E1 -13729.945,E2 -13729.945} C_VEL
LIN {X 0,Y 370.636,Z 258.226,A -85,B 0,C 180,E1 -13731.548,E2 -13731.548} C_VEL
LIN {X 0,Y 378.64,Z 274.99,A -85,B 0,C 180,E1 -13733.009,E2 -13733.009} C_VEL
LIN {X 0,Y 378.926,Z 276.758,A -85,B 0,C 180,E1 -13733.089,E2 -13733.089} C_VEL
LIN {X 0,Y 372.969,Z 435.952,A -85,B 0,C 180,E1 -13736.342,E2 -13736.342} C_VEL
LIN {X 0,Y 371.594,Z 452.458,A -85,B 0,C 180,E1 -13736.859,E2 -13736.859} C_VEL
LIN {X 0,Y 369.953,Z 467.903,A -85,B 0,C 180,E1 -13737.544,E2 -13737.544} C_VEL
LIN {X 0,Y 367.866,Z 483.873,A -85,B 0,C 180,E1 -13738.468,E2 -13738.468} C_VEL
LIN {X 0,Y 365.596,Z 498.602,A -85,B 0,C 180,E1 -13739.535,E2 -13739.535} C_VEL
LIN {X 0,Y 363.012,Z 513.677,A -85,B 0,C 180,E1 -13740.897,E2 -13740.897} C_VEL
LIN {X 0,Y 360.318,Z 527.502,A -85,B 0,C 180,E1 -13742.404,E2 -13742.404} C_VEL
LIN {X 0,Y 357.736,Z 540.365,A -85,B 0,C 180,E1 -13744.081,E2 -13744.081} C_VEL
LIN {X 0,Y 355.14,Z 553.128,A -85,B 0,C 180,E1 -13746.067,E2 -13746.067} C_VEL
LIN {X 0,Y 352.906,Z 564.018,A -85,B 0,C 180,E1 -13748.075,E2 -13748.075} C_VEL
LIN {X 0,Y 350.803,Z 574.21,A -85,B 0,C 180,E1 -13750.321,E2 -13750.321} C_VEL
LIN {X 0,Y 349.356,Z 582.295,A -85,B 0,C 180,E1 -13752.438,E2 -13752.438} C_VEL
LIN {X 0,Y 348.043,Z 589.894,A -85,B 0,C 180,E1 -13754.782,E2 -13754.782} C_VEL
LIN {X 0,Y 347.16,Z 596.121,A -85,B 0,C 180,E1 -13757.134,E2 -13757.134} C_VEL
LIN {X 0,Y 346.514,Z 601.189,A -85,B 0,C 180,E1 -13759.483,E2 -13759.483} C_VEL
LIN {X 0,Y 346.264,Z 605.174,A -85,B 0,C 180,E1 -13761.832,E2 -13761.832} C_VEL
LIN {X 0,Y 346.158,Z 608.068,A -85,B 0,C 180,E1 -13764.174,E2 -13764.174} C_VEL
LIN {X 0,Y 346.114,Z 610.001,A -85,B 0,C 180,E1 -13766.508,E2 -13766.508} C_VEL
LIN {X 0,Y 346.119,Z 610.891,A -85,B 0,C 180,E1 -13768.837,E2 -13768.837} C_VEL
LIN {X 0,Y 346.119,Z 610.859,A -85,B 0,C 180,E1 -13771.164,E2 -13771.164} C_VEL
LIN {X 0,Y 346.114,Z 609.785,A -85,B 0,C 180,E1 -13773.493,E2 -13773.493} C_VEL
LIN {X 0,Y 346.159,Z 607.779,A -85,B 0,C 180,E1 -13775.827,E2 -13775.827} C_VEL
LIN {X 0,Y 346.265,Z 604.674,A -85,B 0,C 180,E1 -13778.168,E2 -13778.168} C_VEL
LIN {X 0,Y 346.497,Z 600.574,A -85,B 0,C 180,E1 -13780.518,E2 -13780.518} C_VEL
LIN {X 0,Y 347.345,Z 593.971,A -85,B 0,C 180,E1 -13783.384,E2 -13783.384} C_VEL
LIN {X 0,Y 348.235,Z 586.894,A -85,B 0,C 180,E1 -13785.81,E2 -13785.81} C_VEL
LIN {X 0,Y 349.642,Z 578.632,A -85,B 0,C 180,E1 -13788.153,E2 -13788.153} C_VEL
LIN {X 0,Y 351.321,Z 568.769,A -85,B 0,C 180,E1 -13790.492,E2 -13790.492} C_VEL
LIN {X 0,Y 353.265,Z 558.621,A -85,B 0,C 180,E1 -13792.518,E2 -13792.518} C_VEL
LIN {X 0,Y 355.543,Z 546.618,A -85,B 0,C 180,E1 -13794.526,E2 -13794.526} C_VEL
LIN {X 0,Y 357.625,Z 535.647,A -85,B 0,C 180,E1 -13796.085,E2 -13796.085} C_VEL
LIN {X 0,Y 359.916,Z 523.006,A -85,B 0,C 180,E1 -13797.63,E2 -13797.63} C_VEL
LIN {X 0,Y 362.414,Z 508.375,A -85,B 0,C 180,E1 -13799.108,E2 -13799.108} C_VEL
LIN {X 0,Y 364.773,Z 492.918,A -85,B 0,C 180,E1 -13800.381,E2 -13800.381} C_VEL
LIN {X 0,Y 366.828,Z 477.621,A -85,B 0,C 180,E1 -13801.391,E2 -13801.391} C_VEL
LIN {X 0,Y 368.602,Z 460.717,A -85,B 0,C 180,E1 -13802.267,E2 -13802.267} C_VEL
LIN {X 0,Y 370.045,Z 445.07,A -85,B 0,C 180,E1 -13802.852,E2 -13802.852} C_VEL
LIN {X 0,Y 371.061,Z 428.264,A -85,B 0,C 180,E1 -13803.276,E2 -13803.276} C_VEL
LIN {X 0,Y 375.999,Z 275.334,A -85,B 0,C 180,E1 -13806.342,E2 -13806.342} C_VEL
LIN {X 0,Y 375.241,Z 272.589,A -85,B 0,C 180,E1 -13806.485,E2 -13806.485} C_VEL
LIN {X 0,Y 364.786,Z 250.794,A -85,B 0,C 180,E1 -13808.16,E2 -13808.16} C_VEL
LIN {X 0,Y 354.546,Z 231.859,A -85,B 0,C 180,E1 -13809.857,E2 -13809.857} C_VEL
LIN {X 0,Y 352.838,Z 228.601,A -85,B 0,C 180,E1 -13810.165,E2 -13810.165} C_VEL
LIN {X 0,Y 347.725,Z 214.476,A -85,B 0,C 180,E1 -13813.261,E2 -13813.261} C_VEL
LIN {X 0,Y 347.722,Z 214.477,A -85,B 0,C 180,E1 -13816.686,E2 -13816.686} C_VEL
LIN {X 0,Y 347.725,Z 214.475,A -85,B 0,C 180,E1 -13820.177,E2 -13820.177} C_VEL
LIN {X 0,Y 347.755,Z 214.469,A -85,B 0,C 180,E1 -13822.679,E2 -13822.679} C_VEL
LIN {X 0,Y 347.746,Z 214.481,A -85,B 0,C 180,E1 -13825.956,E2 -13825.956} C_VEL
LIN {X 0,Y 347.747,Z 214.472,A -85,B 0,C 180,E1 -13829.652,E2 -13829.652} C_VEL
LIN {X 0,Y 347.828,Z 214.448,A -85,B 0,C 180,E1 -13833.608,E2 -13833.608} C_VEL
LIN {X 0,Y 347.786,Z 214.471,A -85,B 0,C 180,E1 -13836.162,E2 -13836.162} C_VEL
LIN {X 0,Y 347.803,Z 214.45,A -85,B 0,C 180,E1 -13839.909,E2 -13839.909} C_VEL
LIN {X 0,Y 347.83,Z 214.468,A -85,B 0,C 180,E1 -13843.568,E2 -13843.568} C_VEL
LIN {X 0,Y 347.887,Z 214.438,A -85,B 0,C 180,E1 -13847.161,E2 -13847.161} C_VEL
LIN {X 0,Y 347.933,Z 214.446,A -85,B 0,C 180,E1 -13850.701,E2 -13850.701} C_VEL
LIN {X 0,Y 348.075,Z 214.438,A -85,B 0,C 180,E1 -13853.042,E2 -13853.042} C_VEL
LIN {X 0,Y 348.202,Z 214.384,A -85,B 0,C 180,E1 -13857.687,E2 -13857.687} C_VEL
LIN {X 0,Y 348.323,Z 214.399,A -85,B 0,C 180,E1 -13860,E2 -13860} C_VEL
LIN {X 0,Y 348.203,Z 214.423,A -85,B 0,C 180,E1 -13862.314,E2 -13862.314} C_VEL
LIN {X 0,Y 348.09,Z 214.432,A -85,B 0,C 180,E1 -13866.958,E2 -13866.958} C_VEL
LIN {X 0,Y 347.926,Z 214.445,A -85,B 0,C 180,E1 -13870.474,E2 -13870.474} C_VEL
LIN {X 0,Y 347.897,Z 214.456,A -85,B 0,C 180,E1 -13874.15,E2 -13874.15} C_VEL
LIN {X 0,Y 347.889,Z 214.44,A -85,B 0,C 180,E1 -13878.29,E2 -13878.29} C_VEL
LIN {X 0,Y 347.787,Z 214.473,A -85,B 0,C 180,E1 -13881.635,E2 -13881.635} C_VEL
LIN {X 0,Y 347.81,Z 214.453,A -85,B 0,C 180,E1 -13885.108,E2 -13885.108} C_VEL
LIN {X 0,Y 347.811,Z 214.468,A -85,B 0,C 180,E1 -13887.694,E2 -13887.694} C_VEL
LIN {X 0,Y 347.763,Z 214.471,A -85,B 0,C 180,E1 -13890.346,E2 -13890.346} C_VEL
LIN {X 0,Y 347.743,Z 214.48,A -85,B 0,C 180,E1 -13894.464,E2 -13894.464} C_VEL
LIN {X 0,Y 347.773,Z 214.46,A -85,B 0,C 180,E1 -13897.989,E2 -13897.989} C_VEL
LIN {X 0,Y 347.749,Z 214.478,A -85,B 0,C 180,E1 -13901.83,E2 -13901.83} C_VEL
LIN {X 0,Y 347.704,Z 214.477,A -85,B 0,C 180,E1 -13905.027,E2 -13905.027} C_VEL
LIN {X 0,Y 347.748,Z 214.47,A -85,B 0,C 180,E1 -13908.397,E2 -13908.397} C_VEL
LIN {X 0,Y 347.772,Z 214.475,A -85,B 0,C 180,E1 -13912.012,E2 -13912.012} C_VEL
LIN {X 0,Y 347.743,Z 214.478,A -85,B 0,C 180,E1 -13915.536,E2 -13915.536} C_VEL
LIN {X 0,Y 347.763,Z 214.473,A -85,B 0,C 180,E1 -13919.654,E2 -13919.654} C_VEL
LIN {X 0,Y 347.85,Z 214.458,A -85,B 0,C 180,E1 -13922.745,E2 -13922.745} C_VEL
LIN {X 0,Y 347.788,Z 214.466,A -85,B 0,C 180,E1 -13926.162,E2 -13926.162} C_VEL
LIN {X 0,Y 347.806,Z 214.449,A -85,B 0,C 180,E1 -13929.909,E2 -13929.909} C_VEL
LIN {X 0,Y 347.866,Z 214.446,A -85,B 0,C 180,E1 -13932.359,E2 -13932.359} C_VEL
LIN {X 0,Y 347.911,Z 214.625,A -85,B 0,C 180,E1 -13935.337,E2 -13935.337} C_VEL
LIN {X 0,Y 348.939,Z 217.338,A -85,B 0,C 180,E1 -13935.545,E2 -13935.545} C_VEL
LIN {X 0,Y 350.741,Z 219.832,A -85,B 0,C 180,E1 -13935.844,E2 -13935.844} C_VEL
LIN {X 0,Y 362.046,Z 238.273,A -85,B 0,C 180,E1 -13937.702,E2 -13937.702} C_VEL
LIN {X 0,Y 370.899,Z 255.099,A -85,B 0,C 180,E1 -13939.12,E2 -13939.12} C_VEL
LIN {X 0,Y 376.144,Z 266.495,A -85,B 0,C 180,E1 -13939.953,E2 -13939.953} C_VEL
LIN {X 0,Y 370.976,Z 417.908,A -85,B 0,C 180,E1 -13942.995,E2 -13942.995} C_VEL
LIN {X 0,Y 369.785,Z 435.197,A -85,B 0,C 180,E1 -13943.555,E2 -13943.555} C_VEL
LIN {X 0,Y 368.237,Z 451.724,A -85,B 0,C 180,E1 -13944.318,E2 -13944.318} C_VEL
LIN {X 0,Y 366.455,Z 467.638,A -85,B 0,C 180,E1 -13945.29,E2 -13945.29} C_VEL
LIN {X 0,Y 364.469,Z 482.343,A -85,B 0,C 180,E1 -13946.407,E2 -13946.407} C_VEL
LIN {X 0,Y 362.429,Z 495.724,A -85,B 0,C 180,E1 -13947.638,E2 -13947.638} C_VEL
LIN {X 0,Y 359.982,Z 509.532,A -85,B 0,C 180,E1 -13949.161,E2 -13949.161} C_VEL
LIN {X 0,Y 357.724,Z 522.051,A -85,B 0,C 180,E1 -13950.816,E2 -13950.816} C_VEL
LIN {X 0,Y 355.555,Z 533.267,A -85,B 0,C 180,E1 -13952.549,E2 -13952.549} C_VEL
LIN {X 0,Y 353.41,Z 544.244,A -85,B 0,C 180,E1 -13954.562,E2 -13954.562} C_VEL
LIN {X 0,Y 351.569,Z 553.63,A -85,B 0,C 180,E1 -13956.6,E2 -13956.6} C_VEL
LIN {X 0,Y 349.89,Z 562.77,A -85,B 0,C 180,E1 -13958.955,E2 -13958.955} C_VEL
LIN {X 0,Y 348.677,Z 569.566,A -85,B 0,C 180,E1 -13961.039,E2 -13961.039} C_VEL
LIN {X 0,Y 347.685,Z 575.804,A -85,B 0,C 180,E1 -13963.358,E2 -13963.358} C_VEL
LIN {X 0,Y 346.917,Z 581.282,A -85,B 0,C 180,E1 -13965.871,E2 -13965.871} C_VEL
LIN {X 0,Y 346.466,Z 584.61,A -85,B 0,C 180,E1 -13967.824,E2 -13967.824} C_VEL
LIN {X 0,Y 345.607,Z 586.04,A -85,B 0,C 180,E1 -13968.767,E2 -13968.767} C_VEL
LIN {X 0,Y 342.507,Z 588.005,A -85,B 0,C 180,E1 -13970.303,E2 -13970.303} C_VEL
LIN {X 0,Y 339.96,Z 589.29,A -85,B 0,C 180,E1 -13971.555,E2 -13971.555} C_VEL
LIN {X 0,Y 338.858,Z 589.995,A -85,B 0,C 180,E1 -13972.532,E2 -13972.532} C_VEL
LIN {X 0,Y 338.76,Z 590.205,A -85,B 0,C 180,E1 -13972.864,E2 -13972.864} C_VEL
LIN {X 0,Y 338.708,Z 590.974,A -85,B 0,C 180,E1 -13974.518,E2 -13974.518} C_VEL
LIN {X 0,Y 338.75,Z 591.173,A -85,B 0,C 180,E1 -13977.156,E2 -13977.156} C_VEL
LIN {X 0,Y 338.864,Z 590.216,A -85,B 0,C 180,E1 -13979.851,E2 -13979.851} C_VEL
LIN {X 0,Y 339.171,Z 587.996,A -85,B 0,C 180,E1 -13982.598,E2 -13982.598} C_VEL
LIN {X 0,Y 339.777,Z 584.32,A -85,B 0,C 180,E1 -13985.39,E2 -13985.39} C_VEL
LIN {X 0,Y 340.561,Z 579.107,A -85,B 0,C 180,E1 -13988.249,E2 -13988.249} C_VEL
LIN {X 0,Y 341.443,Z 574.167,A -85,B 0,C 180,E1 -13990.397,E2 -13990.397} C_VEL
LIN {X 0,Y 342.866,Z 566.909,A -85,B 0,C 180,E1 -13992.964,E2 -13992.964} C_VEL
LIN {X 0,Y 344.783,Z 558.017,A -85,B 0,C 180,E1 -13995.514,E2 -13995.514} C_VEL
LIN {X 0,Y 346.828,Z 548.851,A -85,B 0,C 180,E1 -13997.698,E2 -13997.698} C_VEL
LIN {X 0,Y 349.44,Z 537.616,A -85,B 0,C 180,E1 -13999.94,E2 -13999.94} C_VEL
LIN {X 0,Y 352.001,Z 526.159,A -85,B 0,C 180,E1 -14001.867,E2 -14001.867} C_VEL
LIN {X 0,Y 354.436,Z 514.655,A -85,B 0,C 180,E1 -14003.497,E2 -14003.497} C_VEL
LIN {X 0,Y 357.134,Z 501.29,A -85,B 0,C 180,E1 -14005.093,E2 -14005.093} C_VEL
LIN {X 0,Y 359.56,Z 488.034,A -85,B 0,C 180,E1 -14006.422,E2 -14006.422} C_VEL
LIN {X 0,Y 361.936,Z 473.411,A -85,B 0,C 180,E1 -14007.635,E2 -14007.635} C_VEL
LIN {X 0,Y 364.008,Z 458.194,A -85,B 0,C 180,E1 -14008.646,E2 -14008.646} C_VEL
LIN {X 0,Y 365.794,Z 442.125,A -85,B 0,C 180,E1 -14009.481,E2 -14009.481} C_VEL
LIN {X 0,Y 367.228,Z 425.8,A -85,B 0,C 180,E1 -14010.101,E2 -14010.101} C_VEL
LIN {X 0,Y 368.17,Z 408.713,A -85,B 0,C 180,E1 -14010.539,E2 -14010.539} C_VEL
LIN {X 0,Y 373.468,Z 270.194,A -85,B 0,C 180,E1 -14013.402,E2 -14013.402} C_VEL
LIN {X 0,Y 365.528,Z 254.541,A -85,B 0,C 180,E1 -14014.894,E2 -14014.894} C_VEL
LIN {X 0,Y 356.426,Z 238.805,A -85,B 0,C 180,E1 -14016.687,E2 -14016.687} C_VEL
LIN {X 0,Y 349.467,Z 228.609,A -85,B 0,C 180,E1 -14018.125,E2 -14018.125} C_VEL
LIN {X 0,Y 346.553,Z 224.496,A -85,B 0,C 180,E1 -14018.755,E2 -14018.755} C_VEL
LIN {X 0,Y 344.289,Z 221.191,A -85,B 0,C 180,E1 -14019.265,E2 -14019.265} C_VEL
LIN {X 0,Y 343.546,Z 220.17,A -85,B 0,C 180,E1 -14019.434,E2 -14019.434} C_VEL
LIN {X 0,Y 341.552,Z 217.859,A -85,B 0,C 180,E1 -14019.878,E2 -14019.878} C_VEL
LIN {X 0,Y 340.736,Z 215.349,A -85,B 0,C 180,E1 -14020.142,E2 -14020.142} C_VEL
LIN {X 0,Y 340.769,Z 215.346,A -85,B 0,C 180,E1 -14023.218,E2 -14023.218} C_VEL
LIN {X 0,Y 340.864,Z 215.338,A -85,B 0,C 180,E1 -14025.705,E2 -14025.705} C_VEL
LIN {X 0,Y 340.842,Z 215.335,A -85,B 0,C 180,E1 -14029.305,E2 -14029.305} C_VEL
LIN {X 0,Y 341.039,Z 215.314,A -85,B 0,C 180,E1 -14032.897,E2 -14032.897} C_VEL
LIN {X 0,Y 341.161,Z 215.299,A -85,B 0,C 180,E1 -14037.639,E2 -14037.639} C_VEL
LIN {X 0,Y 341.29,Z 215.284,A -85,B 0,C 180,E1 -14040,E2 -14040} C_VEL
LIN {X 0,Y 341.161,Z 215.299,A -85,B 0,C 180,E1 -14042.361,E2 -14042.361} C_VEL
LIN {X 0,Y 341.054,Z 215.315,A -85,B 0,C 180,E1 -14047.102,E2 -14047.102} C_VEL
LIN {X 0,Y 340.865,Z 215.333,A -85,B 0,C 180,E1 -14050.694,E2 -14050.694} C_VEL
LIN {X 0,Y 340.857,Z 215.336,A -85,B 0,C 180,E1 -14054.325,E2 -14054.325} C_VEL
LIN {X 0,Y 340.831,Z 215.339,A -85,B 0,C 180,E1 -14058.466,E2 -14058.466} C_VEL
LIN {X 0,Y 340.748,Z 215.349,A -85,B 0,C 180,E1 -14061.857,E2 -14061.857} C_VEL
LIN {X 0,Y 340.767,Z 215.352,A -85,B 0,C 180,E1 -14065.665,E2 -14065.665} C_VEL
LIN {X 0,Y 340.723,Z 215.356,A -85,B 0,C 180,E1 -14068.321,E2 -14068.321} C_VEL
LIN {X 0,Y 340.692,Z 215.359,A -85,B 0,C 180,E1 -14071.045,E2 -14071.045} C_VEL
LIN {X 0,Y 340.713,Z 215.361,A -85,B 0,C 180,E1 -14075.279,E2 -14075.279} C_VEL
LIN {X 0,Y 340.705,Z 215.362,A -85,B 0,C 180,E1 -14078.386,E2 -14078.386} C_VEL
LIN {X 0,Y 340.694,Z 215.364,A -85,B 0,C 180,E1 -14082.046,E2 -14082.046} C_VEL
LIN {X 0,Y 340.687,Z 215.494,A -85,B 0,C 180,E1 -14083.601,E2 -14083.601} C_VEL
LIN {X 0,Y 345.441,Z 227.13,A -85,B 0,C 180,E1 -14086.769,E2 -14086.769} C_VEL
LIN {X 0,Y 352.904,Z 238.898,A -85,B 0,C 180,E1 -14088.395,E2 -14088.395} C_VEL
LIN {X 0,Y 360.146,Z 251.339,A -85,B 0,C 180,E1 -14089.878,E2 -14089.878} C_VEL
LIN {X 0,Y 368.053,Z 266.476,A -85,B 0,C 180,E1 -14091.417,E2 -14091.417} C_VEL
LIN {X 0,Y 373.37,Z 277.947,A -85,B 0,C 180,E1 -14092.423,E2 -14092.423} C_VEL
LIN {X 0,Y 367.22,Z 435.611,A -85,B 0,C 180,E1 -14095.693,E2 -14095.693} C_VEL
LIN {X 0,Y 365.791,Z 452.271,A -85,B 0,C 180,E1 -14096.223,E2 -14096.223} C_VEL
LIN {X 0,Y 364.158,Z 467.046,A -85,B 0,C 180,E1 -14096.88,E2 -14096.88} C_VEL
LIN {X 0,Y 362.148,Z 482.176,A -85,B 0,C 180,E1 -14097.747,E2 -14097.747} C_VEL
LIN {X 0,Y 359.748,Z 497.085,A -85,B 0,C 180,E1 -14098.823,E2 -14098.823} C_VEL
LIN {X 0,Y 357.161,Z 511.962,A -85,B 0,C 180,E1 -14100.162,E2 -14100.162} C_VEL
LIN {X 0,Y 354.504,Z 525.231,A -85,B 0,C 180,E1 -14101.589,E2 -14101.589} C_VEL
LIN {X 0,Y 351.751,Z 538.421,A -85,B 0,C 180,E1 -14103.286,E2 -14103.286} C_VEL
LIN {X 0,Y 349.335,Z 549.678,A -85,B 0,C 180,E1 -14105.009,E2 -14105.009} C_VEL
LIN {X 0,Y 346.836,Z 560.967,A -85,B 0,C 180,E1 -14107.042,E2 -14107.042} C_VEL
LIN {X 0,Y 344.484,Z 571.929,A -85,B 0,C 180,E1 -14109.396,E2 -14109.396} C_VEL
LIN {X 0,Y 342.723,Z 581.167,A -85,B 0,C 180,E1 -14111.777,E2 -14111.777} C_VEL
LIN {X 0,Y 341.1,Z 589.765,A -85,B 0,C 180,E1 -14114.464,E2 -14114.464} C_VEL
LIN {X 0,Y 340.162,Z 595.976,A -85,B 0,C 180,E1 -14116.864,E2 -14116.864} C_VEL
LIN {X 0,Y 339.465,Z 601.025,A -85,B 0,C 180,E1 -14119.262,E2 -14119.262} C_VEL
LIN {X 0,Y 339.189,Z 605.005,A -85,B 0,C 180,E1 -14121.661,E2 -14121.661} C_VEL
LIN {X 0,Y 339.061,Z 608.057,A -85,B 0,C 180,E1 -14124.229,E2 -14124.229} C_VEL
LIN {X 0,Y 339.037,Z 609.813,A -85,B 0,C 180,E1 -14126.435,E2 -14126.435} C_VEL
LIN {X 0,Y 339.02,Z 610.688,A -85,B 0,C 180,E1 -14128.813,E2 -14128.813} C_VEL
LIN {X 0,Y 339.021,Z 610.65,A -85,B 0,C 180,E1 -14131.188,E2 -14131.188} C_VEL
LIN {X 0,Y 339.038,Z 609.561,A -85,B 0,C 180,E1 -14133.566,E2 -14133.566} C_VEL
LIN {X 0,Y 339.084,Z 607.546,A -85,B 0,C 180,E1 -14135.949,E2 -14135.949} C_VEL
LIN {X 0,Y 339.19,Z 604.422,A -85,B 0,C 180,E1 -14138.34,E2 -14138.34} C_VEL
LIN {X 0,Y 339.446,Z 600.305,A -85,B 0,C 180,E1 -14140.739,E2 -14140.739} C_VEL
LIN {X 0,Y 340.171,Z 594.965,A -85,B 0,C 180,E1 -14143.136,E2 -14143.136} C_VEL
LIN {X 0,Y 341.013,Z 588.427,A -85,B 0,C 180,E1 -14145.541,E2 -14145.541} C_VEL
LIN {X 0,Y 342.416,Z 580.566,A -85,B 0,C 180,E1 -14147.931,E2 -14147.931} C_VEL
LIN {X 0,Y 344.062,Z 571.067,A -85,B 0,C 180,E1 -14150.319,E2 -14150.319} C_VEL
LIN {X 0,Y 345.993,Z 561.259,A -85,B 0,C 180,E1 -14152.387,E2 -14152.387} C_VEL
LIN {X 0,Y 348.257,Z 550.089,A -85,B 0,C 180,E1 -14154.387,E2 -14154.387} C_VEL
LIN {X 0,Y 350.464,Z 538.368,A -85,B 0,C 180,E1 -14156.179,E2 -14156.179} C_VEL
LIN {X 0,Y 353.077,Z 524.883,A -85,B 0,C 180,E1 -14157.889,E2 -14157.889} C_VEL
LIN {X 0,Y 355.453,Z 511.626,A -85,B 0,C 180,E1 -14159.298,E2 -14159.298} C_VEL
LIN {X 0,Y 357.774,Z 497.543,A -85,B 0,C 180,E1 -14160.549,E2 -14160.549} C_VEL
LIN {X 0,Y 360.02,Z 482.395,A -85,B 0,C 180,E1 -14161.643,E2 -14161.643} C_VEL
LIN {X 0,Y 361.842,Z 466.851,A -85,B 0,C 180,E1 -14162.532,E2 -14162.532} C_VEL
LIN {X 0,Y 363.359,Z 451.367,A -85,B 0,C 180,E1 -14163.203,E2 -14163.203} C_VEL
LIN {X 0,Y 364.647,Z 435.268,A -85,B 0,C 180,E1 -14163.691,E2 -14163.691} C_VEL
LIN {X 0,Y 370.127,Z 276.646,A -85,B 0,C 180,E1 -14166.932,E2 -14166.932} C_VEL
LIN {X 0,Y 360.207,Z 255.638,A -85,B 0,C 180,E1 -14168.567,E2 -14168.567} C_VEL
LIN {X 0,Y 349.663,Z 236.012,A -85,B 0,C 180,E1 -14170.359,E2 -14170.359} C_VEL
LIN {X 0,Y 345.374,Z 228.219,A -85,B 0,C 180,E1 -14171.157,E2 -14171.157} C_VEL
LIN {X 0,Y 340.639,Z 215.367,A -85,B 0,C 180,E1 -14174.044,E2 -14174.044} C_VEL
LIN {X 0,Y 340.694,Z 215.36,A -85,B 0,C 180,E1 -14177.955,E2 -14177.955} C_VEL
LIN {X 0,Y 340.718,Z 215.358,A -85,B 0,C 180,E1 -14181.771,E2 -14181.771} C_VEL
LIN {X 0,Y 340.721,Z 215.357,A -85,B 0,C 180,E1 -14185.595,E2 -14185.595} C_VEL
LIN {X 0,Y 340.695,Z 215.341,A -85,B 0,C 180,E1 -14188.955,E2 -14188.955} C_VEL
LIN {X 0,Y 340.774,Z 215.339,A -85,B 0,C 180,E1 -14192.475,E2 -14192.475} C_VEL
LIN {X 0,Y 340.754,Z 215.343,A -85,B 0,C 180,E1 -14195.638,E2 -14195.638} C_VEL
LIN {X 0,Y 340.738,Z 215.335,A -85,B 0,C 180,E1 -14199.474,E2 -14199.474} C_VEL
LIN {X 0,Y 340.79,Z 215.328,A -85,B 0,C 180,E1 -14201.981,E2 -14201.981} C_VEL
LIN {X 0,Y 340.868,Z 215.333,A -85,B 0,C 180,E1 -14205.705,E2 -14205.705} C_VEL
LIN {X 0,Y 340.845,Z 215.31,A -85,B 0,C 180,E1 -14209.305,E2 -14209.305} C_VEL
LIN {X 0,Y 341.043,Z 215.314,A -85,B 0,C 180,E1 -14212.898,E2 -14212.898} C_VEL
LIN {X 0,Y 341.164,Z 215.259,A -85,B 0,C 180,E1 -14217.639,E2 -14217.639} C_VEL
LIN {X 0,Y 341.274,Z 215.277,A -85,B 0,C 180,E1 -14220,E2 -14220} C_VEL
LIN {X 0,Y 341.165,Z 215.299,A -85,B 0,C 180,E1 -14222.361,E2 -14222.361} C_VEL
LIN {X 0,Y 341.058,Z 215.308,A -85,B 0,C 180,E1 -14227.102,E2 -14227.102} C_VEL
LIN {X 0,Y 340.868,Z 215.322,A -85,B 0,C 180,E1 -14230.694,E2 -14230.694} C_VEL
LIN {X 0,Y 340.861,Z 215.335,A -85,B 0,C 180,E1 -14234.325,E2 -14234.325} C_VEL
LIN {X 0,Y 340.835,Z 215.318,A -85,B 0,C 180,E1 -14238.466,E2 -14238.466} C_VEL
LIN {X 0,Y 340.752,Z 215.352,A -85,B 0,C 180,E1 -14241.857,E2 -14241.857} C_VEL
LIN {X 0,Y 340.771,Z 215.329,A -85,B 0,C 180,E1 -14245.664,E2 -14245.664} C_VEL
LIN {X 0,Y 340.741,Z 215.353,A -85,B 0,C 180,E1 -14248.32,E2 -14248.32} C_VEL
LIN {X 0,Y 340.703,Z 215.345,A -85,B 0,C 180,E1 -14251.044,E2 -14251.044} C_VEL
LIN {X 0,Y 340.717,Z 215.357,A -85,B 0,C 180,E1 -14255.279,E2 -14255.279} C_VEL
LIN {X 0,Y 340.709,Z 215.34,A -85,B 0,C 180,E1 -14258.386,E2 -14258.386} C_VEL
LIN {X 0,Y 340.697,Z 215.354,A -85,B 0,C 180,E1 -14262.045,E2 -14262.045} C_VEL
LIN {X 0,Y 340.65,Z 215.364,A -85,B 0,C 180,E1 -14266.227,E2 -14266.227} C_VEL
LIN {X 0,Y 340.686,Z 215.35,A -85,B 0,C 180,E1 -14269.753,E2 -14269.753} C_VEL
LIN {X 0,Y 340.703,Z 215.346,A -85,B 0,C 180,E1 -14273.258,E2 -14273.258} C_VEL
LIN {X 0,Y 340.691,Z 215.36,A -85,B 0,C 180,E1 -14276.153,E2 -14276.153} C_VEL
LIN {X 0,Y 340.774,Z 215.349,A -85,B 0,C 180,E1 -14280.332,E2 -14280.332} C_VEL
LIN {X 0,Y 340.803,Z 215.336,A -85,B 0,C 180,E1 -14283.02,E2 -14283.02} C_VEL
LIN {X 0,Y 340.729,Z 215.347,A -85,B 0,C 180,E1 -14286.927,E2 -14286.927} C_VEL
LIN {X 0,Y 340.786,Z 215.315,A -85,B 0,C 180,E1 -14290.733,E2 -14290.733} C_VEL
LIN {X 0,Y 340.793,Z 215.352,A -85,B 0,C 180,E1 -14293.835,E2 -14293.835} C_VEL
LIN {X 0,Y 340.803,Z 215.339,A -85,B 0,C 180,E1 -14294.373,E2 -14294.373} C_VEL
LIN {X 0,Y 341.951,Z 218.398,A -85,B 0,C 180,E1 -14294.644,E2 -14294.644} C_VEL
LIN {X 0,Y 343.557,Z 220.408,A -85,B 0,C 180,E1 -14294.916,E2 -14294.916} C_VEL
LIN {X 0,Y 345.738,Z 223.808,A -85,B 0,C 180,E1 -14295.299,E2 -14295.299} C_VEL
LIN {X 0,Y 357.577,Z 243.255,A -85,B 0,C 180,E1 -14297.302,E2 -14297.302} C_VEL
LIN {X 0,Y 366.11,Z 259.618,A -85,B 0,C 180,E1 -14298.7,E2 -14298.7} C_VEL
LIN {X 0,Y 370.179,Z 268.398,A -85,B 0,C 180,E1 -14299.363,E2 -14299.363} C_VEL
LIN {X 0,Y 364.915,Z 418.301,A -85,B 0,C 180,E1 -14302.426,E2 -14302.426} C_VEL
LIN {X 0,Y 363.767,Z 434.598,A -85,B 0,C 180,E1 -14302.96,E2 -14302.96} C_VEL
LIN {X 0,Y 362.159,Z 451.36,A -85,B 0,C 180,E1 -14303.733,E2 -14303.733} C_VEL
LIN {X 0,Y 360.338,Z 466.953,A -85,B 0,C 180,E1 -14304.684,E2 -14304.684} C_VEL
LIN {X 0,Y 358.358,Z 481.425,A -85,B 0,C 180,E1 -14305.782,E2 -14305.782} C_VEL
LIN {X 0,Y 356.16,Z 494.967,A -85,B 0,C 180,E1 -14307.031,E2 -14307.031} C_VEL
LIN {X 0,Y 353.687,Z 508.903,A -85,B 0,C 180,E1 -14308.576,E2 -14308.576} C_VEL
LIN {X 0,Y 351.197,Z 522.293,A -85,B 0,C 180,E1 -14310.364,E2 -14310.364} C_VEL
LIN {X 0,Y 348.694,Z 534.558,A -85,B 0,C 180,E1 -14312.31,E2 -14312.31} C_VEL
LIN {X 0,Y 346.483,Z 545.444,A -85,B 0,C 180,E1 -14314.362,E2 -14314.362} C_VEL
LIN {X 0,Y 344.396,Z 555.919,A -85,B 0,C 180,E1 -14316.738,E2 -14316.738} C_VEL
LIN {X 0,Y 342.666,Z 564.706,A -85,B 0,C 180,E1 -14319.146,E2 -14319.146} C_VEL
LIN {X 0,Y 341.485,Z 571.224,A -85,B 0,C 180,E1 -14321.274,E2 -14321.274} C_VEL
LIN {X 0,Y 340.353,Z 577.957,A -85,B 0,C 180,E1 -14323.95,E2 -14323.95} C_VEL
LIN {X 0,Y 339.607,Z 583.541,A -85,B 0,C 180,E1 -14326.841,E2 -14326.841} C_VEL
LIN {X 0,Y 339.131,Z 587.087,A -85,B 0,C 180,E1 -14329.364,E2 -14329.364} C_VEL
LIN {X 0,Y 338.849,Z 589.582,A -85,B 0,C 180,E1 -14331.921,E2 -14331.921} C_VEL
LIN {X 0,Y 338.76,Z 590.205,A -85,B 0,C 180,E1 -14332.864,E2 -14332.864} C_VEL
LIN {X 0,Y 338.06,Z 590.786,A -85,B 0,C 180,E1 -14333.852,E2 -14333.852} C_VEL
LIN {X 0,Y 335.175,Z 591.376,A -85,B 0,C 180,E1 -14335.464,E2 -14335.464} C_VEL
LIN {X 0,Y 332.762,Z 591.471,A -85,B 0,C 180,E1 -14336.771,E2 -14336.771} C_VEL
LIN {X 0,Y 331.745,Z 591.311,A -85,B 0,C 180,E1 -14337.782,E2 -14337.782} C_VEL
LIN {X 0,Y 331.672,Z 591.195,A -85,B 0,C 180,E1 -14338.125,E2 -14338.125} C_VEL
LIN {X 0,Y 331.834,Z 590.05,A -85,B 0,C 180,E1 -14340.55,E2 -14340.55} C_VEL
LIN {X 0,Y 332.217,Z 587.514,A -85,B 0,C 180,E1 -14343.368,E2 -14343.368} C_VEL
LIN {X 0,Y 332.737,Z 584.696,A -85,B 0,C 180,E1 -14345.509,E2 -14345.509} C_VEL
LIN {X 0,Y 333.471,Z 579.907,A -85,B 0,C 180,E1 -14348.25,E2 -14348.25} C_VEL
LIN {X 0,Y 334.613,Z 574.008,A -85,B 0,C 180,E1 -14350.877,E2 -14350.877} C_VEL
LIN {X 0,Y 335.935,Z 567.577,A -85,B 0,C 180,E1 -14353.198,E2 -14353.198} C_VEL
LIN {X 0,Y 337.655,Z 560.001,A -85,B 0,C 180,E1 -14355.469,E2 -14355.469} C_VEL
LIN {X 0,Y 339.744,Z 551.117,A -85,B 0,C 180,E1 -14357.723,E2 -14357.723} C_VEL
LIN {X 0,Y 342.243,Z 540.904,A -85,B 0,C 180,E1 -14359.885,E2 -14359.885} C_VEL
LIN {X 0,Y 344.929,Z 529.617,A -85,B 0,C 180,E1 -14361.891,E2 -14361.891} C_VEL
LIN {X 0,Y 347.63,Z 517.472,A -85,B 0,C 180,E1 -14363.72,E2 -14363.72} C_VEL
LIN {X 0,Y 350.369,Z 504.79,A -85,B 0,C 180,E1 -14365.325,E2 -14365.325} C_VEL
LIN {X 0,Y 353.282,Z 489.826,A -85,B 0,C 180,E1 -14366.896,E2 -14366.896} C_VEL
LIN {X 0,Y 355.963,Z 474.085,A -85,B 0,C 180,E1 -14368.233,E2 -14368.233} C_VEL
LIN {X 0,Y 358.153,Z 458.631,A -85,B 0,C 180,E1 -14369.282,E2 -14369.282} C_VEL
LIN {X 0,Y 359.964,Z 443.027,A -85,B 0,C 180,E1 -14370.109,E2 -14370.109} C_VEL
LIN {X 0,Y 361.464,Z 426.617,A -85,B 0,C 180,E1 -14370.75,E2 -14370.75} C_VEL
LIN {X 0,Y 362.521,Z 408.903,A -85,B 0,C 180,E1 -14371.208,E2 -14371.208} C_VEL
LIN {X 0,Y 368.02,Z 272.763,A -85,B 0,C 180,E1 -14374.057,E2 -14374.057} C_VEL
LIN {X 0,Y 359.923,Z 256.869,A -85,B 0,C 180,E1 -14375.635,E2 -14375.635} C_VEL
LIN {X 0,Y 351.511,Z 242.391,A -85,B 0,C 180,E1 -14377.364,E2 -14377.364} C_VEL
LIN {X 0,Y 345.407,Z 233.525,A -85,B 0,C 180,E1 -14378.672,E2 -14378.672} C_VEL
LIN {X 0,Y 342.419,Z 229.317,A -85,B 0,C 180,E1 -14379.343,E2 -14379.343} C_VEL
LIN {X 0,Y 339.887,Z 225.664,A -85,B 0,C 180,E1 -14379.933,E2 -14379.933} C_VEL
LIN {X 0,Y 337.632,Z 222.64,A -85,B 0,C 180,E1 -14380.467,E2 -14380.467} C_VEL
LIN {X 0,Y 336.77,Z 221.238,A -85,B 0,C 180,E1 -14380.685,E2 -14380.685} C_VEL
LIN {X 0,Y 334.708,Z 219.042,A -85,B 0,C 180,E1 -14381.173,E2 -14381.173} C_VEL
LIN {X 0,Y 333.81,Z 216.704,A -85,B 0,C 180,E1 -14381.438,E2 -14381.438} C_VEL
LIN {X 0,Y 333.742,Z 216.218,A -85,B 0,C 180,E1 -14381.485,E2 -14381.485} C_VEL
LIN {X 0,Y 333.802,Z 216.215,A -85,B 0,C 180,E1 -14385.577,E2 -14385.577} C_VEL
LIN {X 0,Y 333.811,Z 216.206,A -85,B 0,C 180,E1 -14389.077,E2 -14389.077} C_VEL
LIN {X 0,Y 333.986,Z 216.193,A -85,B 0,C 180,E1 -14392.747,E2 -14392.747} C_VEL
LIN {X 0,Y 333.799,Z 216.216,A -85,B 0,C 180,E1 -14395.169,E2 -14395.169} C_VEL
LIN {X 0,Y 334.099,Z 216.179,A -85,B 0,C 180,E1 -14397.589,E2 -14397.589} C_VEL
LIN {X 0,Y 334.241,Z 216.161,A -85,B 0,C 180,E1 -14400,E2 -14400} C_VEL
LIN {X 0,Y 334.099,Z 216.178,A -85,B 0,C 180,E1 -14402.411,E2 -14402.411} C_VEL
LIN {X 0,Y 334.009,Z 216.188,A -85,B 0,C 180,E1 -14406.039,E2 -14406.039} C_VEL
LIN {X 0,Y 333.953,Z 216.195,A -85,B 0,C 180,E1 -14408.471,E2 -14408.471} C_VEL
LIN {X 0,Y 333.786,Z 216.22,A -85,B 0,C 180,E1 -14412.155,E2 -14412.155} C_VEL
LIN {X 0,Y 333.772,Z 216.218,A -85,B 0,C 180,E1 -14415.886,E2 -14415.886} C_VEL
LIN {X 0,Y 333.79,Z 216.215,A -85,B 0,C 180,E1 -14418.655,E2 -14418.655} C_VEL
LIN {X 0,Y 333.687,Z 216.23,A -85,B 0,C 180,E1 -14422.278,E2 -14422.278} C_VEL
LIN {X 0,Y 333.73,Z 216.223,A -85,B 0,C 180,E1 -14426.247,E2 -14426.247} C_VEL
LIN {X 0,Y 333.685,Z 216.23,A -85,B 0,C 180,E1 -14428.974,E2 -14428.974} C_VEL
LIN {X 0,Y 333.638,Z 216.242,A -85,B 0,C 180,E1 -14432.587,E2 -14432.587} C_VEL
LIN {X 0,Y 333.671,Z 216.236,A -85,B 0,C 180,E1 -14436.139,E2 -14436.139} C_VEL
LIN {X 0,Y 333.642,Z 216.247,A -85,B 0,C 180,E1 -14439.193,E2 -14439.193} C_VEL
LIN {X 0,Y 333.643,Z 216.283,A -85,B 0,C 180,E1 -14442.33,E2 -14442.33} C_VEL
LIN {X 0,Y 337.933,Z 226.775,A -85,B 0,C 180,E1 -14445.369,E2 -14445.369} C_VEL
LIN {X 0,Y 345.458,Z 238.254,A -85,B 0,C 180,E1 -14447.123,E2 -14447.123} C_VEL
LIN {X 0,Y 353.619,Z 251.897,A -85,B 0,C 180,E1 -14448.893,E2 -14448.893} C_VEL
LIN {X 0,Y 362.588,Z 268.945,A -85,B 0,C 180,E1 -14450.722,E2 -14450.722} C_VEL
LIN {X 0,Y 367.808,Z 280.327,A -85,B 0,C 180,E1 -14451.753,E2 -14451.753} C_VEL
LIN {X 0,Y 363.529,Z 385.722,A -85,B 0,C 180,E1 -14453.955,E2 -14453.955} C_VEL
LIN {X 0,Y 361.469,Z 436.257,A -85,B 0,C 180,E1 -14455.045,E2 -14455.045} C_VEL
LIN {X 0,Y 359.856,Z 454.057,A -85,B 0,C 180,E1 -14455.631,E2 -14455.631} C_VEL
LIN {X 0,Y 358.099,Z 468.891,A -85,B 0,C 180,E1 -14456.329,E2 -14456.329} C_VEL
LIN {X 0,Y 355.872,Z 484.492,A -85,B 0,C 180,E1 -14457.275,E2 -14457.275} C_VEL
LIN {X 0,Y 353.399,Z 498.992,A -85,B 0,C 180,E1 -14458.365,E2 -14458.365} C_VEL
LIN {X 0,Y 350.695,Z 513.523,A -85,B 0,C 180,E1 -14459.72,E2 -14459.72} C_VEL
LIN {X 0,Y 347.994,Z 526.486,A -85,B 0,C 180,E1 -14461.173,E2 -14461.173} C_VEL
LIN {X 0,Y 345.387,Z 538.452,A -85,B 0,C 180,E1 -14462.753,E2 -14462.753} C_VEL
LIN {X 0,Y 342.817,Z 549.691,A -85,B 0,C 180,E1 -14464.5,E2 -14464.5} C_VEL
LIN {X 0,Y 340.221,Z 560.934,A -85,B 0,C 180,E1 -14466.569,E2 -14466.569} C_VEL
LIN {X 0,Y 337.743,Z 571.85,A -85,B 0,C 180,E1 -14468.965,E2 -14468.965} C_VEL
LIN {X 0,Y 335.885,Z 581.059,A -85,B 0,C 180,E1 -14471.393,E2 -14471.393} C_VEL
LIN {X 0,Y 334.159,Z 589.639,A -85,B 0,C 180,E1 -14474.133,E2 -14474.133} C_VEL
LIN {X 0,Y 333.162,Z 595.843,A -85,B 0,C 180,E1 -14476.583,E2 -14476.583} C_VEL
LIN {X 0,Y 332.429,Z 600.873,A -85,B 0,C 180,E1 -14479.032,E2 -14479.032} C_VEL
LIN {X 0,Y 332.098,Z 604.841,A -85,B 0,C 180,E1 -14481.482,E2 -14481.482} C_VEL
LIN {X 0,Y 331.984,Z 608.015,A -85,B 0,C 180,E1 -14484.251,E2 -14484.251} C_VEL
LIN {X 0,Y 331.94,Z 609.625,A -85,B 0,C 180,E1 -14486.359,E2 -14486.359} C_VEL
LIN {X 0,Y 331.925,Z 610.486,A -85,B 0,C 180,E1 -14488.787,E2 -14488.787} C_VEL
LIN {X 0,Y 331.926,Z 610.441,A -85,B 0,C 180,E1 -14491.214,E2 -14491.214} C_VEL
LIN {X 0,Y 331.962,Z 609.336,A -85,B 0,C 180,E1 -14493.642,E2 -14493.642} C_VEL
LIN {X 0,Y 331.991,Z 607.312,A -85,B 0,C 180,E1 -14496.076,E2 -14496.076} C_VEL
LIN {X 0,Y 332.098,Z 604.169,A -85,B 0,C 180,E1 -14498.519,E2 -14498.519} C_VEL
LIN {X 0,Y 332.411,Z 600.034,A -85,B 0,C 180,E1 -14500.969,E2 -14500.969} C_VEL
LIN {X 0,Y 333.156,Z 594.681,A -85,B 0,C 180,E1 -14503.418,E2 -14503.418} C_VEL
LIN {X 0,Y 334.054,Z 588.115,A -85,B 0,C 180,E1 -14505.873,E2 -14505.873} C_VEL
LIN {X 0,Y 335.547,Z 580.223,A -85,B 0,C 180,E1 -14508.311,E2 -14508.311} C_VEL
LIN {X 0,Y 337.293,Z 570.695,A -85,B 0,C 180,E1 -14510.746,E2 -14510.746} C_VEL
LIN {X 0,Y 339.315,Z 560.843,A -85,B 0,C 180,E1 -14512.852,E2 -14512.852} C_VEL
LIN {X 0,Y 341.794,Z 549.044,A -85,B 0,C 180,E1 -14514.984,E2 -14514.984} C_VEL
LIN {X 0,Y 344.283,Z 536.805,A -85,B 0,C 180,E1 -14516.849,E2 -14516.849} C_VEL
LIN {X 0,Y 346.974,Z 523.147,A -85,B 0,C 180,E1 -14518.589,E2 -14518.589} C_VEL
LIN {X 0,Y 349.72,Z 508.127,A -85,B 0,C 180,E1 -14520.159,E2 -14520.159} C_VEL
LIN {X 0,Y 352.171,Z 493.269,A -85,B 0,C 180,E1 -14521.423,E2 -14521.423} C_VEL
LIN {X 0,Y 354.373,Z 478.182,A -85,B 0,C 180,E1 -14522.46,E2 -14522.46} C_VEL
LIN {X 0,Y 356.22,Z 462.381,A -85,B 0,C 180,E1 -14523.322,E2 -14523.322} C_VEL
LIN {X 0,Y 357.777,Z 446.491,A -85,B 0,C 180,E1 -14523.96,E2 -14523.96} C_VEL
LIN {X 0,Y 358.943,Z 428.946,A -85,B 0,C 180,E1 -14524.427,E2 -14524.427} C_VEL
LIN {X 0,Y 364.205,Z 278.631,A -85,B 0,C 180,E1 -14527.536,E2 -14527.536} C_VEL
LIN {X 0,Y 354.731,Z 258.793,A -85,B 0,C 180,E1 -14529.134,E2 -14529.134} C_VEL
LIN {X 0,Y 344.727,Z 240.004,A -85,B 0,C 180,E1 -14530.89,E2 -14530.89} C_VEL
LIN {X 0,Y 337.948,Z 228.05,A -85,B 0,C 180,E1 -14532.154,E2 -14532.154} C_VEL
LIN {X 0,Y 333.583,Z 216.238,A -85,B 0,C 180,E1 -14534.953,E2 -14534.953} C_VEL
LIN {X 0,Y 333.638,Z 216.241,A -85,B 0,C 180,E1 -14537.618,E2 -14537.618} C_VEL
LIN {X 0,Y 333.638,Z 216.242,A -85,B 0,C 180,E1 -14541.205,E2 -14541.205} C_VEL
LIN {X 0,Y 333.673,Z 216.217,A -85,B 0,C 180,E1 -14543.861,E2 -14543.861} C_VEL
LIN {X 0,Y 333.641,Z 216.224,A -85,B 0,C 180,E1 -14547.413,E2 -14547.413} C_VEL
LIN {X 0,Y 333.688,Z 216.235,A -85,B 0,C 180,E1 -14551.026,E2 -14551.026} C_VEL
LIN {X 0,Y 333.733,Z 216.202,A -85,B 0,C 180,E1 -14553.754,E2 -14553.754} C_VEL
LIN {X 0,Y 333.718,Z 216.229,A -85,B 0,C 180,E1 -14557.914,E2 -14557.914} C_VEL
LIN {X 0,Y 333.738,Z 216.2,A -85,B 0,C 180,E1 -14561.586,E2 -14561.586} C_VEL
LIN {X 0,Y 333.806,Z 216.213,A -85,B 0,C 180,E1 -14565.577,E2 -14565.577} C_VEL
LIN {X 0,Y 333.815,Z 216.183,A -85,B 0,C 180,E1 -14569.077,E2 -14569.077} C_VEL
LIN {X 0,Y 333.99,Z 216.194,A -85,B 0,C 180,E1 -14572.747,E2 -14572.747} C_VEL
LIN {X 0,Y 333.801,Z 216.195,A -85,B 0,C 180,E1 -14575.169,E2 -14575.169} C_VEL
LIN {X 0,Y 334.101,Z 216.138,A -85,B 0,C 180,E1 -14577.589,E2 -14577.589} C_VEL
LIN {X 0,Y 334.225,Z 216.155,A -85,B 0,C 180,E1 -14580,E2 -14580} C_VEL
LIN {X 0,Y 334.102,Z 216.178,A -85,B 0,C 180,E1 -14582.411,E2 -14582.411} C_VEL
LIN {X 0,Y 333.99,Z 216.179,A -85,B 0,C 180,E1 -14586.663,E2 -14586.663} C_VEL
LIN {X 0,Y 333.849,Z 216.208,A -85,B 0,C 180,E1 -14589.695,E2 -14589.695} C_VEL
LIN {X 0,Y 333.794,Z 216.205,A -85,B 0,C 180,E1 -14593.391,E2 -14593.391} C_VEL
LIN {X 0,Y 333.745,Z 216.216,A -85,B 0,C 180,E1 -14597.146,E2 -14597.146} C_VEL
LIN {X 0,Y 333.734,Z 216.206,A -85,B 0,C 180,E1 -14599.69,E2 -14599.69} C_VEL
LIN {X 0,Y 333.691,Z 216.231,A -85,B 0,C 180,E1 -14602.278,E2 -14602.278} C_VEL
LIN {X 0,Y 333.734,Z 216.208,A -85,B 0,C 180,E1 -14606.246,E2 -14606.246} C_VEL
LIN {X 0,Y 333.71,Z 216.228,A -85,B 0,C 180,E1 -14608.972,E2 -14608.972} C_VEL
LIN {X 0,Y 333.644,Z 216.22,A -85,B 0,C 180,E1 -14612.588,E2 -14612.588} C_VEL
LIN {X 0,Y 333.675,Z 216.229,A -85,B 0,C 180,E1 -14616.139,E2 -14616.139} C_VEL
LIN {X 0,Y 333.645,Z 216.224,A -85,B 0,C 180,E1 -14619.192,E2 -14619.192} C_VEL
LIN {X 0,Y 333.631,Z 216.233,A -85,B 0,C 180,E1 -14622.5,E2 -14622.5} C_VEL
LIN {X 0,Y 333.595,Z 216.245,A -85,B 0,C 180,E1 -14625.955,E2 -14625.955} C_VEL
LIN {X 0,Y 333.646,Z 216.224,A -85,B 0,C 180,E1 -14629.315,E2 -14629.315} C_VEL
LIN {X 0,Y 333.664,Z 216.223,A -85,B 0,C 180,E1 -14633.168,E2 -14633.168} C_VEL
LIN {X 0,Y 333.673,Z 216.228,A -85,B 0,C 180,E1 -14635.341,E2 -14635.341} C_VEL
LIN {X 0,Y 333.702,Z 216.225,A -85,B 0,C 180,E1 -14639.71,E2 -14639.71} C_VEL
LIN {X 0,Y 333.742,Z 216.216,A -85,B 0,C 180,E1 -14642.401,E2 -14642.401} C_VEL
LIN {X 0,Y 333.727,Z 216.226,A -85,B 0,C 180,E1 -14645.091,E2 -14645.091} C_VEL
LIN {X 0,Y 333.677,Z 216.223,A -85,B 0,C 180,E1 -14649.019,E2 -14649.019} C_VEL
LIN {X 0,Y 333.792,Z 216.187,A -85,B 0,C 180,E1 -14651.589,E2 -14651.589} C_VEL
LIN {X 0,Y 333.757,Z 216.261,A -85,B 0,C 180,E1 -14653.439,E2 -14653.439} C_VEL
LIN {X 0,Y 334.763,Z 219.072,A -85,B 0,C 180,E1 -14653.665,E2 -14653.665} C_VEL
LIN {X 0,Y 336.624,Z 221.582,A -85,B 0,C 180,E1 -14654,E2 -14654} C_VEL
LIN {X 0,Y 346.215,Z 236.569,A -85,B 0,C 180,E1 -14655.708,E2 -14655.708} C_VEL
LIN {X 0,Y 353.832,Z 249.588,A -85,B 0,C 180,E1 -14657.014,E2 -14657.014} C_VEL
LIN {X 0,Y 361.514,Z 264.555,A -85,B 0,C 180,E1 -14658.302,E2 -14658.302} C_VEL
LIN {X 0,Y 364.331,Z 270.655,A -85,B 0,C 180,E1 -14658.772,E2 -14658.772} C_VEL
LIN {X 0,Y 358.886,Z 418.698,A -85,B 0,C 180,E1 -14661.838,E2 -14661.838} C_VEL
LIN {X 0,Y 357.635,Z 435.813,A -85,B 0,C 180,E1 -14662.413,E2 -14662.413} C_VEL
LIN {X 0,Y 355.965,Z 452.297,A -85,B 0,C 180,E1 -14663.196,E2 -14663.196} C_VEL
LIN {X 0,Y 354.094,Z 467.712,A -85,B 0,C 180,E1 -14664.162,E2 -14664.162} C_VEL
LIN {X 0,Y 351.978,Z 482.394,A -85,B 0,C 180,E1 -14665.303,E2 -14665.303} C_VEL
LIN {X 0,Y 349.588,Z 496.953,A -85,B 0,C 180,E1 -14666.686,E2 -14666.686} C_VEL
LIN {X 0,Y 346.964,Z 510.636,A -85,B 0,C 180,E1 -14668.259,E2 -14668.259} C_VEL
LIN {X 0,Y 344.528,Z 523.235,A -85,B 0,C 180,E1 -14670,E2 -14670} C_VEL
LIN {X 0,Y 341.836,Z 535.832,A -85,B 0,C 180,E1 -14672.062,E2 -14672.062} C_VEL
LIN {X 0,Y 339.568,Z 546.546,A -85,B 0,C 180,E1 -14674.154,E2 -14674.154} C_VEL
LIN {X 0,Y 337.43,Z 556.911,A -85,B 0,C 180,E1 -14676.577,E2 -14676.577} C_VEL
LIN {X 0,Y 335.658,Z 565.589,A -85,B 0,C 180,E1 -14679.034,E2 -14679.034} C_VEL
LIN {X 0,Y 334.287,Z 572.81,A -85,B 0,C 180,E1 -14681.52,E2 -14681.52} C_VEL
LIN {X 0,Y 333.244,Z 578.798,A -85,B 0,C 180,E1 -14684.041,E2 -14684.041} C_VEL
LIN {X 0,Y 332.583,Z 583.565,A -85,B 0,C 180,E1 -14686.575,E2 -14686.575} C_VEL
LIN {X 0,Y 332.171,Z 586.393,A -85,B 0,C 180,E1 -14688.503,E2 -14688.503} C_VEL
LIN {X 0,Y 331.838,Z 589.336,A -85,B 0,C 180,E1 -14691.271,E2 -14691.271} C_VEL
LIN {X 0,Y 331.624,Z 591.098,A -85,B 0,C 180,E1 -14694.317,E2 -14694.317} C_VEL
LIN {X 0,Y 331.653,Z 591.39,A -85,B 0,C 180,E1 -14697.125,E2 -14697.125} C_VEL
LIN {X 0,Y 331.672,Z 591.195,A -85,B 0,C 180,E1 -14698.125,E2 -14698.125} C_VEL
LIN {X 0,Y 331.045,Z 590.88,A -85,B 0,C 180,E1 -14699.137,E2 -14699.137} C_VEL
LIN {X 0,Y 328.299,Z 590.047,A -85,B 0,C 180,E1 -14700.787,E2 -14700.787} C_VEL
LIN {X 0,Y 326.032,Z 589.103,A -85,B 0,C 180,E1 -14702.118,E2 -14702.118} C_VEL
LIN {X 0,Y 325.156,Z 588.206,A -85,B 0,C 180,E1 -14703.139,E2 -14703.139} C_VEL
LIN {X 0,Y 325.136,Z 587.789,A -85,B 0,C 180,E1 -14703.482,E2 -14703.482} C_VEL
LIN {X 0,Y 325.675,Z 585.07,A -85,B 0,C 180,E1 -14705.637,E2 -14705.637} C_VEL
LIN {X 0,Y 326.518,Z 579.981,A -85,B 0,C 180,E1 -14708.622,E2 -14708.622} C_VEL
LIN {X 0,Y 327.787,Z 573.866,A -85,B 0,C 180,E1 -14711.373,E2 -14711.373} C_VEL
LIN {X 0,Y 329.408,Z 566.648,A -85,B 0,C 180,E1 -14713.992,E2 -14713.992} C_VEL
LIN {X 0,Y 331.533,Z 557.942,A -85,B 0,C 180,E1 -14716.555,E2 -14716.555} C_VEL
LIN {X 0,Y 333.832,Z 548.684,A -85,B 0,C 180,E1 -14718.817,E2 -14718.817} C_VEL
LIN {X 0,Y 336.457,Z 538.239,A -85,B 0,C 180,E1 -14720.971,E2 -14720.971} C_VEL
LIN {X 0,Y 339.098,Z 527.677,A -85,B 0,C 180,E1 -14722.819,E2 -14722.819} C_VEL
LIN {X 0,Y 342.018,Z 515.194,A -85,B 0,C 180,E1 -14724.657,E2 -14724.657} C_VEL
LIN {X 0,Y 345.026,Z 501.311,A -85,B 0,C 180,E1 -14726.365,E2 -14726.365} C_VEL
LIN {X 0,Y 347.81,Z 487.245,A -85,B 0,C 180,E1 -14727.795,E2 -14727.795} C_VEL
LIN {X 0,Y 350.295,Z 473.269,A -85,B 0,C 180,E1 -14728.969,E2 -14728.969} C_VEL
LIN {X 0,Y 352.633,Z 457.071,A -85,B 0,C 180,E1 -14730.062,E2 -14730.062} C_VEL
LIN {X 0,Y 354.517,Z 441.109,A -85,B 0,C 180,E1 -14730.884,E2 -14730.884} C_VEL
LIN {X 0,Y 355.997,Z 424.579,A -85,B 0,C 180,E1 -14731.504,E2 -14731.504} C_VEL
LIN {X 0,Y 357.149,Z 403.17,A -85,B 0,C 180,E1 -14732.027,E2 -14732.027} C_VEL
LIN {X 0,Y 362.612,Z 275.82,A -85,B 0,C 180,E1 -14734.723,E2 -14734.723} C_VEL
LIN {X 0,Y 360.99,Z 271.941,A -85,B 0,C 180,E1 -14735.06,E2 -14735.06} C_VEL
LIN {X 0,Y 353.586,Z 257.806,A -85,B 0,C 180,E1 -14736.576,E2 -14736.576} C_VEL
LIN {X 0,Y 347.32,Z 247.081,A -85,B 0,C 180,E1 -14737.92,E2 -14737.92} C_VEL
LIN {X 0,Y 341.722,Z 238.851,A -85,B 0,C 180,E1 -14739.162,E2 -14739.162} C_VEL
LIN {X 0,Y 336.349,Z 231.156,A -85,B 0,C 180,E1 -14740.429,E2 -14740.429} C_VEL
LIN {X 0,Y 333.088,Z 226.725,A -85,B 0,C 180,E1 -14741.235,E2 -14741.235} C_VEL
LIN {X 0,Y 330.793,Z 223.678,A -85,B 0,C 180,E1 -14741.817,E2 -14741.817} C_VEL
LIN {X 0,Y 330.076,Z 222.322,A -85,B 0,C 180,E1 -14742.017,E2 -14742.017} C_VEL
LIN {X 0,Y 327.861,Z 220.243,A -85,B 0,C 180,E1 -14742.577,E2 -14742.577} C_VEL
LIN {X 0,Y 326.757,Z 217.654,A -85,B 0,C 180,E1 -14742.919,E2 -14742.919} C_VEL
LIN {X 0,Y 326.674,Z 217.104,A -85,B 0,C 180,E1 -14742.995,E2 -14742.995} C_VEL
LIN {X 0,Y 326.753,Z 217.097,A -85,B 0,C 180,E1 -14746.314,E2 -14746.314} C_VEL
LIN {X 0,Y 326.777,Z 217.094,A -85,B 0,C 180,E1 -14750.093,E2 -14750.093} C_VEL
LIN {X 0,Y 326.975,Z 217.065,A -85,B 0,C 180,E1 -14753.831,E2 -14753.831} C_VEL
LIN {X 0,Y 327.039,Z 217.058,A -85,B 0,C 180,E1 -14757.537,E2 -14757.537} C_VEL
LIN {X 0,Y 327.192,Z 217.039,A -85,B 0,C 180,E1 -14760,E2 -14760} C_VEL
LIN {X 0,Y 327.04,Z 217.057,A -85,B 0,C 180,E1 -14762.463,E2 -14762.463} C_VEL
LIN {X 0,Y 326.984,Z 217.063,A -85,B 0,C 180,E1 -14766.169,E2 -14766.169} C_VEL
LIN {X 0,Y 326.8,Z 217.092,A -85,B 0,C 180,E1 -14769.907,E2 -14769.907} C_VEL
LIN {X 0,Y 326.753,Z 217.091,A -85,B 0,C 180,E1 -14773.686,E2 -14773.686} C_VEL
LIN {X 0,Y 326.694,Z 217.103,A -85,B 0,C 180,E1 -14777.528,E2 -14777.528} C_VEL
LIN {X 0,Y 326.657,Z 217.109,A -85,B 0,C 180,E1 -14780.135,E2 -14780.135} C_VEL
LIN {X 0,Y 326.647,Z 217.105,A -85,B 0,C 180,E1 -14784.129,E2 -14784.129} C_VEL
LIN {X 0,Y 326.677,Z 217.1,A -85,B 0,C 180,E1 -14786.858,E2 -14786.858} C_VEL
LIN {X 0,Y 326.629,Z 217.114,A -85,B 0,C 180,E1 -14790.61,E2 -14790.61} C_VEL
LIN {X 0,Y 326.602,Z 217.115,A -85,B 0,C 180,E1 -14794.02,E2 -14794.02} C_VEL
LIN {X 0,Y 326.623,Z 217.119,A -85,B 0,C 180,E1 -14797.239,E2 -14797.239} C_VEL
LIN {X 0,Y 326.624,Z 217.211,A -85,B 0,C 180,E1 -14800.988,E2 -14800.988} C_VEL
LIN {X 0,Y 330.456,Z 226.383,A -85,B 0,C 180,E1 -14803.845,E2 -14803.845} C_VEL
LIN {X 0,Y 338.7,Z 238.74,A -85,B 0,C 180,E1 -14805.912,E2 -14805.912} C_VEL
LIN {X 0,Y 345.417,Z 249.677,A -85,B 0,C 180,E1 -14807.473,E2 -14807.473} C_VEL
LIN {X 0,Y 352.123,Z 261.674,A -85,B 0,C 180,E1 -14808.944,E2 -14808.944} C_VEL
LIN {X 0,Y 359.088,Z 275.43,A -85,B 0,C 180,E1 -14810.4,E2 -14810.4} C_VEL
LIN {X 0,Y 362.372,Z 282.671,A -85,B 0,C 180,E1 -14811.068,E2 -14811.068} C_VEL
LIN {X 0,Y 357.808,Z 389.438,A -85,B 0,C 180,E1 -14813.329,E2 -14813.329} C_VEL
LIN {X 0,Y 355.854,Z 435.872,A -85,B 0,C 180,E1 -14814.349,E2 -14814.349} C_VEL
LIN {X 0,Y 354.233,Z 453.179,A -85,B 0,C 180,E1 -14814.919,E2 -14814.919} C_VEL
LIN {X 0,Y 352.404,Z 468.188,A -85,B 0,C 180,E1 -14815.624,E2 -14815.624} C_VEL
LIN {X 0,Y 350.256,Z 482.915,A -85,B 0,C 180,E1 -14816.511,E2 -14816.511} C_VEL
LIN {X 0,Y 347.672,Z 497.66,A -85,B 0,C 180,E1 -14817.611,E2 -14817.611} C_VEL
LIN {X 0,Y 344.826,Z 512.595,A -85,B 0,C 180,E1 -14819.013,E2 -14819.013} C_VEL
LIN {X 0,Y 342.016,Z 525.424,A -85,B 0,C 180,E1 -14820.452,E2 -14820.452} C_VEL
LIN {X 0,Y 339.035,Z 538.486,A -85,B 0,C 180,E1 -14822.199,E2 -14822.199} C_VEL
LIN {X 0,Y 336.047,Z 551.015,A -85,B 0,C 180,E1 -14824.197,E2 -14824.197} C_VEL
LIN {X 0,Y 333.286,Z 562.408,A -85,B 0,C 180,E1 -14826.382,E2 -14826.382} C_VEL
LIN {X 0,Y 331.027,Z 571.796,A -85,B 0,C 180,E1 -14828.517,E2 -14828.517} C_VEL
LIN {X 0,Y 329.046,Z 580.969,A -85,B 0,C 180,E1 -14830.991,E2 -14830.991} C_VEL
LIN {X 0,Y 327.219,Z 589.513,A -85,B 0,C 180,E1 -14833.787,E2 -14833.787} C_VEL
LIN {X 0,Y 326.156,Z 595.709,A -85,B 0,C 180,E1 -14836.289,E2 -14836.289} C_VEL
LIN {X 0,Y 325.407,Z 600.721,A -85,B 0,C 180,E1 -14838.792,E2 -14838.792} C_VEL
LIN {X 0,Y 325.028,Z 604.682,A -85,B 0,C 180,E1 -14841.295,E2 -14841.295} C_VEL
LIN {X 0,Y 324.888,Z 608.01,A -85,B 0,C 180,E1 -14844.308,E2 -14844.308} C_VEL
LIN {X 0,Y 324.846,Z 609.441,A -85,B 0,C 180,E1 -14846.279,E2 -14846.279} C_VEL
LIN {X 0,Y 324.833,Z 610.285,A -85,B 0,C 180,E1 -14848.761,E2 -14848.761} C_VEL
LIN {X 0,Y 324.834,Z 610.232,A -85,B 0,C 180,E1 -14851.24,E2 -14851.24} C_VEL
LIN {X 0,Y 324.866,Z 609.109,A -85,B 0,C 180,E1 -14853.721,E2 -14853.721} C_VEL
LIN {X 0,Y 324.89,Z 607.072,A -85,B 0,C 180,E1 -14856.21,E2 -14856.21} C_VEL
LIN {X 0,Y 325.026,Z 603.91,A -85,B 0,C 180,E1 -14858.706,E2 -14858.706} C_VEL
LIN {X 0,Y 325.39,Z 599.751,A -85,B 0,C 180,E1 -14861.209,E2 -14861.209} C_VEL
LIN {X 0,Y 326.159,Z 594.38,A -85,B 0,C 180,E1 -14863.711,E2 -14863.711} C_VEL
LIN {X 0,Y 327.137,Z 587.786,A -85,B 0,C 180,E1 -14866.218,E2 -14866.218} C_VEL
LIN {X 0,Y 328.67,Z 579.861,A -85,B 0,C 180,E1 -14868.708,E2 -14868.708} C_VEL
LIN {X 0,Y 330.536,Z 570.316,A -85,B 0,C 180,E1 -14871.19,E2 -14871.19} C_VEL
LIN {X 0,Y 332.97,Z 558.915,A -85,B 0,C 180,E1 -14873.643,E2 -14873.643} C_VEL
LIN {X 0,Y 335.259,Z 548.442,A -85,B 0,C 180,E1 -14875.532,E2 -14875.532} C_VEL
LIN {X 0,Y 337.864,Z 536.293,A -85,B 0,C 180,E1 -14877.402,E2 -14877.402} C_VEL
LIN {X 0,Y 340.642,Z 522.582,A -85,B 0,C 180,E1 -14879.171,E2 -14879.171} C_VEL
LIN {X 0,Y 343.509,Z 507.51,A -85,B 0,C 180,E1 -14880.763,E2 -14880.763} C_VEL
LIN {X 0,Y 346.069,Z 492.545,A -85,B 0,C 180,E1 -14882.042,E2 -14882.042} C_VEL
LIN {X 0,Y 348.335,Z 477.297,A -85,B 0,C 180,E1 -14883.094,E2 -14883.094} C_VEL
LIN {X 0,Y 350.279,Z 460.471,A -85,B 0,C 180,E1 -14884.006,E2 -14884.006} C_VEL
LIN {X 0,Y 351.866,Z 444.873,A -85,B 0,C 180,E1 -14884.615,E2 -14884.615} C_VEL
LIN {X 0,Y 353,Z 428.029,A -85,B 0,C 180,E1 -14885.058,E2 -14885.058} C_VEL
LIN {X 0,Y 358.387,Z 280.971,A -85,B 0,C 180,E1 -14888.136,E2 -14888.136} C_VEL
LIN {X 0,Y 349.541,Z 262.395,A -85,B 0,C 180,E1 -14889.674,E2 -14889.674} C_VEL
LIN {X 0,Y 340.149,Z 244.629,A -85,B 0,C 180,E1 -14891.367,E2 -14891.367} C_VEL
LIN {X 0,Y 331.654,Z 229.907,A -85,B 0,C 180,E1 -14892.972,E2 -14892.972} C_VEL
LIN {X 0,Y 330.432,Z 227.559,A -85,B 0,C 180,E1 -14893.276,E2 -14893.276} C_VEL
LIN {X 0,Y 326.566,Z 217.107,A -85,B 0,C 180,E1 -14895.849,E2 -14895.849} C_VEL
LIN {X 0,Y 326.583,Z 217.105,A -85,B 0,C 180,E1 -14899.79,E2 -14899.79} C_VEL
LIN {X 0,Y 326.624,Z 217.097,A -85,B 0,C 180,E1 -14902.953,E2 -14902.953} C_VEL
LIN {X 0,Y 326.605,Z 217.115,A -85,B 0,C 180,E1 -14905.981,E2 -14905.981} C_VEL
LIN {X 0,Y 326.646,Z 217.106,A -85,B 0,C 180,E1 -14910.34,E2 -14910.34} C_VEL
LIN {X 0,Y 326.688,Z 217.079,A -85,B 0,C 180,E1 -14914.516,E2 -14914.516} C_VEL
LIN {X 0,Y 326.642,Z 217.102,A -85,B 0,C 180,E1 -14918.545,E2 -14918.545} C_VEL
LIN {X 0,Y 326.705,Z 217.072,A -85,B 0,C 180,E1 -14921.175,E2 -14921.175} C_VEL
LIN {X 0,Y 326.761,Z 217.091,A -85,B 0,C 180,E1 -14925.433,E2 -14925.433} C_VEL
LIN {X 0,Y 326.756,Z 217.059,A -85,B 0,C 180,E1 -14928.839,E2 -14928.839} C_VEL
LIN {X 0,Y 326.94,Z 217.074,A -85,B 0,C 180,E1 -14932.59,E2 -14932.59} C_VEL
LIN {X 0,Y 326.979,Z 217.063,A -85,B 0,C 180,E1 -14933.831,E2 -14933.831} C_VEL
LIN {X 0,Y 327.042,Z 217.015,A -85,B 0,C 180,E1 -14937.537,E2 -14937.537} C_VEL
LIN {X 0,Y 327.177,Z 217.032,A -85,B 0,C 180,E1 -14940,E2 -14940} C_VEL
LIN {X 0,Y 327.043,Z 217.057,A -85,B 0,C 180,E1 -14942.463,E2 -14942.463} C_VEL
LIN {X 0,Y 326.957,Z 217.054,A -85,B 0,C 180,E1 -14946.655,E2 -14946.655} C_VEL
LIN {X 0,Y 326.804,Z 217.082,A -85,B 0,C 180,E1 -14949.907,E2 -14949.907} C_VEL
LIN {X 0,Y 326.757,Z 217.084,A -85,B 0,C 180,E1 -14953.685,E2 -14953.685} C_VEL
LIN {X 0,Y 326.697,Z 217.086,A -85,B 0,C 180,E1 -14957.528,E2 -14957.528} C_VEL
LIN {X 0,Y 326.661,Z 217.091,A -85,B 0,C 180,E1 -14960.135,E2 -14960.135} C_VEL
LIN {X 0,Y 326.65,Z 217.094,A -85,B 0,C 180,E1 -14964.129,E2 -14964.129} C_VEL
LIN {X 0,Y 326.684,Z 217.093,A -85,B 0,C 180,E1 -14966.858,E2 -14966.858} C_VEL
LIN {X 0,Y 326.638,Z 217.101,A -85,B 0,C 180,E1 -14970.611,E2 -14970.611} C_VEL
LIN {X 0,Y 326.606,Z 217.11,A -85,B 0,C 180,E1 -14974.019,E2 -14974.019} C_VEL
LIN {X 0,Y 326.626,Z 217.098,A -85,B 0,C 180,E1 -14977.239,E2 -14977.239} C_VEL
LIN {X 0,Y 326.577,Z 217.118,A -85,B 0,C 180,E1 -14981.131,E2 -14981.131} C_VEL
LIN {X 0,Y 326.526,Z 217.113,A -85,B 0,C 180,E1 -14984.743,E2 -14984.743} C_VEL
LIN {X 0,Y 326.575,Z 217.108,A -85,B 0,C 180,E1 -14988.154,E2 -14988.154} C_VEL
LIN {X 0,Y 326.622,Z 217.114,A -85,B 0,C 180,E1 -14991.391,E2 -14991.391} C_VEL
LIN {X 0,Y 326.618,Z 217.102,A -85,B 0,C 180,E1 -14994.851,E2 -14994.851} C_VEL
LIN {X 0,Y 326.607,Z 217.108,A -85,B 0,C 180,E1 -14997.456,E2 -14997.456} C_VEL
LIN {X 0,Y 326.66,Z 217.108,A -85,B 0,C 180,E1 -15000.341,E2 -15000.341} C_VEL
LIN {X 0,Y 326.69,Z 217.104,A -85,B 0,C 180,E1 -15004.516,E2 -15004.516} C_VEL
LIN {X 0,Y 326.644,Z 217.107,A -85,B 0,C 180,E1 -15008.545,E2 -15008.545} C_VEL
LIN {X 0,Y 326.717,Z 217.073,A -85,B 0,C 180,E1 -15012.15,E2 -15012.15} C_VEL
LIN {X 0,Y 326.726,Z 217.076,A -85,B 0,C 180,E1 -15012.393,E2 -15012.393} C_VEL
LIN {X 0,Y 327.709,Z 219.931,A -85,B 0,C 180,E1 -15012.653,E2 -15012.653} C_VEL
LIN {X 0,Y 329.521,Z 222.211,A -85,B 0,C 180,E1 -15012.992,E2 -15012.992} C_VEL
LIN {X 0,Y 331.726,Z 225.674,A -85,B 0,C 180,E1 -15013.418,E2 -15013.418} C_VEL
LIN {X 0,Y 341.693,Z 241.3,A -85,B 0,C 180,E1 -15015.244,E2 -15015.244} C_VEL
LIN {X 0,Y 349.31,Z 254.394,A -85,B 0,C 180,E1 -15016.581,E2 -15016.581} C_VEL
LIN {X 0,Y 356.83,Z 269.288,A -85,B 0,C 180,E1 -15017.88,E2 -15017.88} C_VEL
LIN {X 0,Y 358.499,Z 272.982,A -85,B 0,C 180,E1 -15018.168,E2 -15018.168} C_VEL
LIN {X 0,Y 352.88,Z 418.917,A -85,B 0,C 180,E1 -15021.229,E2 -15021.229} C_VEL
LIN {X 0,Y 351.59,Z 436.031,A -85,B 0,C 180,E1 -15021.812,E2 -15021.812} C_VEL
LIN {X 0,Y 349.932,Z 451.889,A -85,B 0,C 180,E1 -15022.571,E2 -15022.571} C_VEL
LIN {X 0,Y 347.87,Z 468.432,A -85,B 0,C 180,E1 -15023.62,E2 -15023.62} C_VEL
LIN {X 0,Y 345.636,Z 483.266,A -85,B 0,C 180,E1 -15024.8,E2 -15024.8} C_VEL
LIN {X 0,Y 343.191,Z 497.548,A -85,B 0,C 180,E1 -15026.184,E2 -15026.184} C_VEL
LIN {X 0,Y 340.272,Z 512.351,A -85,B 0,C 180,E1 -15027.928,E2 -15027.928} C_VEL
LIN {X 0,Y 337.343,Z 526.666,A -85,B 0,C 180,E1 -15030,E2 -15030} C_VEL
LIN {X 0,Y 334.64,Z 538.746,A -85,B 0,C 180,E1 -15032.106,E2 -15032.106} C_VEL
LIN {X 0,Y 332.339,Z 549.02,A -85,B 0,C 180,E1 -15034.244,E2 -15034.244} C_VEL
LIN {X 0,Y 330.199,Z 558.996,A -85,B 0,C 180,E1 -15036.722,E2 -15036.722} C_VEL
LIN {X 0,Y 328.453,Z 567.318,A -85,B 0,C 180,E1 -15039.207,E2 -15039.207} C_VEL
LIN {X 0,Y 327.081,Z 574.391,A -85,B 0,C 180,E1 -15041.778,E2 -15041.778} C_VEL
LIN {X 0,Y 326.125,Z 579.615,A -85,B 0,C 180,E1 -15044.129,E2 -15044.129} C_VEL
LIN {X 0,Y 325.552,Z 583.578,A -85,B 0,C 180,E1 -15046.298,E2 -15046.298} C_VEL
LIN {X 0,Y 324.999,Z 587.239,A -85,B 0,C 180,E1 -15048.927,E2 -15048.927} C_VEL
LIN {X 0,Y 324.712,Z 589.845,A -85,B 0,C 180,E1 -15051.588,E2 -15051.588} C_VEL
LIN {X 0,Y 324.515,Z 591.397,A -85,B 0,C 180,E1 -15054.552,E2 -15054.552} C_VEL
LIN {X 0,Y 324.558,Z 591.572,A -85,B 0,C 180,E1 -15057.4,E2 -15057.4} C_VEL
LIN {X 0,Y 324.718,Z 590.664,A -85,B 0,C 180,E1 -15060.034,E2 -15060.034} C_VEL
LIN {X 0,Y 325.022,Z 588.626,A -85,B 0,C 180,E1 -15062.722,E2 -15062.722} C_VEL
LIN {X 0,Y 325.136,Z 587.789,A -85,B 0,C 180,E1 -15063.482,E2 -15063.482} C_VEL
LIN {X 0,Y 324.678,Z 586.698,A -85,B 0,C 180,E1 -15064.5,E2 -15064.5} C_VEL
LIN {X 0,Y 322.214,Z 584.62,A -85,B 0,C 180,E1 -15066.163,E2 -15066.163} C_VEL
LIN {X 0,Y 320.183,Z 582.708,A -85,B 0,C 180,E1 -15067.496,E2 -15067.496} C_VEL
LIN {X 0,Y 319.492,Z 581.024,A -85,B 0,C 180,E1 -15068.508,E2 -15068.508} C_VEL
LIN {X 0,Y 319.535,Z 580.381,A -85,B 0,C 180,E1 -15068.845,E2 -15068.845} C_VEL
LIN {X 0,Y 320.566,Z 575.611,A -85,B 0,C 180,E1 -15071.124,E2 -15071.124} C_VEL
LIN {X 0,Y 322.306,Z 568.154,A -85,B 0,C 180,E1 -15073.981,E2 -15073.981} C_VEL
LIN {X 0,Y 324.466,Z 559.659,A -85,B 0,C 180,E1 -15076.614,E2 -15076.614} C_VEL
LIN {X 0,Y 327.161,Z 549.434,A -85,B 0,C 180,E1 -15079.219,E2 -15079.219} C_VEL
LIN {X 0,Y 330.024,Z 538.658,A -85,B 0,C 180,E1 -15081.498,E2 -15081.498} C_VEL
LIN {X 0,Y 333.034,Z 527.166,A -85,B 0,C 180,E1 -15083.535,E2 -15083.535} C_VEL
LIN {X 0,Y 335.938,Z 515.271,A -85,B 0,C 180,E1 -15085.301,E2 -15085.301} C_VEL
LIN {X 0,Y 338.774,Z 502.66,A -85,B 0,C 180,E1 -15086.885,E2 -15086.885} C_VEL
LIN {X 0,Y 341.653,Z 488.89,A -85,B 0,C 180,E1 -15088.33,E2 -15088.33} C_VEL
LIN {X 0,Y 344.378,Z 474.159,A -85,B 0,C 180,E1 -15089.599,E2 -15089.599} C_VEL
LIN {X 0,Y 346.706,Z 458.998,A -85,B 0,C 180,E1 -15090.648,E2 -15090.648} C_VEL
LIN {X 0,Y 348.704,Z 442.976,A -85,B 0,C 180,E1 -15091.515,E2 -15091.515} C_VEL
LIN {X 0,Y 350.288,Z 426.827,A -85,B 0,C 180,E1 -15092.154,E2 -15092.154} C_VEL
LIN {X 0,Y 351.359,Z 409.874,A -85,B 0,C 180,E1 -15092.61,E2 -15092.61} C_VEL
LIN {X 0,Y 357.232,Z 277.881,A -85,B 0,C 180,E1 -15095.44,E2 -15095.44} C_VEL
LIN {X 0,Y 350.526,Z 264.623,A -85,B 0,C 180,E1 -15096.86,E2 -15096.86} C_VEL
LIN {X 0,Y 343.59,Z 252.386,A -85,B 0,C 180,E1 -15098.397,E2 -15098.397} C_VEL
LIN {X 0,Y 335.835,Z 240.798,A -85,B 0,C 180,E1 -15100.202,E2 -15100.202} C_VEL
LIN {X 0,Y 329.759,Z 232.387,A -85,B 0,C 180,E1 -15101.723,E2 -15101.723} C_VEL
LIN {X 0,Y 327.14,Z 228.69,A -85,B 0,C 180,E1 -15102.423,E2 -15102.423} C_VEL
LIN {X 0,Y 324.163,Z 225.128,A -85,B 0,C 180,E1 -15103.225,E2 -15103.225} C_VEL
LIN {X 0,Y 323.001,Z 223.141,A -85,B 0,C 180,E1 -15103.569,E2 -15103.569} C_VEL
LIN {X 0,Y 320.818,Z 221.047,A -85,B 0,C 180,E1 -15104.173,E2 -15104.173} C_VEL
LIN {X 0,Y 319.786,Z 218.574,A -85,B 0,C 180,E1 -15104.525,E2 -15104.525} C_VEL
LIN {X 0,Y 319.679,Z 217.964,A -85,B 0,C 180,E1 -15104.63,E2 -15104.63} C_VEL
LIN {X 0,Y 319.675,Z 217.964,A -85,B 0,C 180,E1 -15107.3,E2 -15107.3} C_VEL
LIN {X 0,Y 319.823,Z 217.956,A -85,B 0,C 180,E1 -15111.432,E2 -15111.432} C_VEL
LIN {X 0,Y 319.929,Z 217.942,A -85,B 0,C 180,E1 -15113.694,E2 -15113.694} C_VEL
LIN {X 0,Y 319.983,Z 217.937,A -85,B 0,C 180,E1 -15117.482,E2 -15117.482} C_VEL
LIN {X 0,Y 320.144,Z 217.917,A -85,B 0,C 180,E1 -15120,E2 -15120} C_VEL
LIN {X 0,Y 319.983,Z 217.936,A -85,B 0,C 180,E1 -15122.518,E2 -15122.518} C_VEL
LIN {X 0,Y 319.938,Z 217.942,A -85,B 0,C 180,E1 -15126.306,E2 -15126.306} C_VEL
LIN {X 0,Y 319.832,Z 217.954,A -85,B 0,C 180,E1 -15128.848,E2 -15128.848} C_VEL
LIN {X 0,Y 319.676,Z 217.977,A -85,B 0,C 180,E1 -15132.7,E2 -15132.7} C_VEL
LIN {X 0,Y 319.694,Z 217.976,A -85,B 0,C 180,E1 -15135.296,E2 -15135.296} C_VEL
LIN {X 0,Y 319.669,Z 217.973,A -85,B 0,C 180,E1 -15139.255,E2 -15139.255} C_VEL
LIN {X 0,Y 319.565,Z 217.992,A -85,B 0,C 180,E1 -15143.32,E2 -15143.32} C_VEL
LIN {X 0,Y 319.629,Z 217.981,A -85,B 0,C 180,E1 -15146.088,E2 -15146.088} C_VEL
LIN {X 0,Y 319.574,Z 217.987,A -85,B 0,C 180,E1 -15148.935,E2 -15148.935} C_VEL
LIN {X 0,Y 319.525,Z 217.996,A -85,B 0,C 180,E1 -15151.862,E2 -15151.862} C_VEL
LIN {X 0,Y 319.575,Z 217.992,A -85,B 0,C 180,E1 -15155.543,E2 -15155.543} C_VEL
LIN {X 0,Y 319.577,Z 218.053,A -85,B 0,C 180,E1 -15159.49,E2 -15159.49} C_VEL
LIN {X 0,Y 322.964,Z 225.978,A -85,B 0,C 180,E1 -15162.168,E2 -15162.168} C_VEL
LIN {X 0,Y 328.545,Z 234.194,A -85,B 0,C 180,E1 -15163.722,E2 -15163.722} C_VEL
LIN {X 0,Y 334.941,Z 243.856,A -85,B 0,C 180,E1 -15165.364,E2 -15165.364} C_VEL
LIN {X 0,Y 342.8,Z 256.788,A -85,B 0,C 180,E1 -15167.241,E2 -15167.241} C_VEL
LIN {X 0,Y 351.469,Z 273.247,A -85,B 0,C 180,E1 -15169.181,E2 -15169.181} C_VEL
LIN {X 0,Y 357.011,Z 285.203,A -85,B 0,C 180,E1 -15170.372,E2 -15170.372} C_VEL
LIN {X 0,Y 350.379,Z 434.533,A -85,B 0,C 180,E1 -15173.603,E2 -15173.603} C_VEL
LIN {X 0,Y 348.737,Z 451.636,A -85,B 0,C 180,E1 -15174.155,E2 -15174.155} C_VEL
LIN {X 0,Y 346.753,Z 467.534,A -85,B 0,C 180,E1 -15174.894,E2 -15174.894} C_VEL
LIN {X 0,Y 344.38,Z 483.306,A -85,B 0,C 180,E1 -15175.861,E2 -15175.861} C_VEL
LIN {X 0,Y 341.696,Z 497.955,A -85,B 0,C 180,E1 -15176.973,E2 -15176.973} C_VEL
LIN {X 0,Y 338.613,Z 513.46,A -85,B 0,C 180,E1 -15178.458,E2 -15178.458} C_VEL
LIN {X 0,Y 335.557,Z 526.745,A -85,B 0,C 180,E1 -15179.998,E2 -15179.998} C_VEL
LIN {X 0,Y 332.715,Z 538.575,A -85,B 0,C 180,E1 -15181.624,E2 -15181.624} C_VEL
LIN {X 0,Y 329.817,Z 550.195,A -85,B 0,C 180,E1 -15183.504,E2 -15183.504} C_VEL
LIN {X 0,Y 326.727,Z 562.387,A -85,B 0,C 180,E1 -15185.878,E2 -15185.878} C_VEL
LIN {X 0,Y 324.046,Z 572.989,A -85,B 0,C 180,E1 -15188.365,E2 -15188.365} C_VEL
LIN {X 0,Y 322.027,Z 581.91,A -85,B 0,C 180,E1 -15190.892,E2 -15190.892} C_VEL
LIN {X 0,Y 320.325,Z 589.409,A -85,B 0,C 180,E1 -15193.428,E2 -15193.428} C_VEL
LIN {X 0,Y 319.173,Z 595.585,A -85,B 0,C 180,E1 -15195.983,E2 -15195.983} C_VEL
LIN {X 0,Y 318.39,Z 600.572,A -85,B 0,C 180,E1 -15198.542,E2 -15198.542} C_VEL
LIN {X 0,Y 317.943,Z 604.524,A -85,B 0,C 180,E1 -15201.099,E2 -15201.099} C_VEL
LIN {X 0,Y 317.802,Z 607.99,A -85,B 0,C 180,E1 -15204.35,E2 -15204.35} C_VEL
LIN {X 0,Y 317.756,Z 609.256,A -85,B 0,C 180,E1 -15206.196,E2 -15206.196} C_VEL
LIN {X 0,Y 317.744,Z 610.083,A -85,B 0,C 180,E1 -15208.733,E2 -15208.733} C_VEL
LIN {X 0,Y 317.745,Z 610.02,A -85,B 0,C 180,E1 -15211.268,E2 -15211.268} C_VEL
LIN {X 0,Y 317.773,Z 608.879,A -85,B 0,C 180,E1 -15213.805,E2 -15213.805} C_VEL
LIN {X 0,Y 317.804,Z 606.827,A -85,B 0,C 180,E1 -15216.349,E2 -15216.349} C_VEL
LIN {X 0,Y 317.939,Z 603.646,A -85,B 0,C 180,E1 -15218.902,E2 -15218.902} C_VEL
LIN {X 0,Y 318.372,Z 599.464,A -85,B 0,C 180,E1 -15221.46,E2 -15221.46} C_VEL
LIN {X 0,Y 319.32,Z 593.113,A -85,B 0,C 180,E1 -15224.441,E2 -15224.441} C_VEL
LIN {X 0,Y 320.555,Z 585.614,A -85,B 0,C 180,E1 -15227.216,E2 -15227.216} C_VEL
LIN {X 0,Y 322.027,Z 578.362,A -85,B 0,C 180,E1 -15229.44,E2 -15229.44} C_VEL
LIN {X 0,Y 324.081,Z 568.597,A -85,B 0,C 180,E1 -15231.968,E2 -15231.968} C_VEL
LIN {X 0,Y 326.358,Z 558.498,A -85,B 0,C 180,E1 -15234.152,E2 -15234.152} C_VEL
LIN {X 0,Y 328.78,Z 547.651,A -85,B 0,C 180,E1 -15236.131,E2 -15236.131} C_VEL
LIN {X 0,Y 331.648,Z 534.661,A -85,B 0,C 180,E1 -15238.132,E2 -15238.132} C_VEL
LIN {X 0,Y 334.342,Z 521.95,A -85,B 0,C 180,E1 -15239.776,E2 -15239.776} C_VEL
LIN {X 0,Y 337.354,Z 506.805,A -85,B 0,C 180,E1 -15241.387,E2 -15241.387} C_VEL
LIN {X 0,Y 340.029,Z 491.736,A -85,B 0,C 180,E1 -15242.682,E2 -15242.682} C_VEL
LIN {X 0,Y 342.321,Z 476.314,A -85,B 0,C 180,E1 -15243.752,E2 -15243.752} C_VEL
LIN {X 0,Y 344.284,Z 459.99,A -85,B 0,C 180,E1 -15244.638,E2 -15244.638} C_VEL
LIN {X 0,Y 345.889,Z 444.157,A -85,B 0,C 180,E1 -15245.261,E2 -15245.261} C_VEL
LIN {X 0,Y 347.072,Z 427.031,A -85,B 0,C 180,E1 -15245.71,E2 -15245.71} C_VEL
LIN {X 0,Y 352.548,Z 283.144,A -85,B 0,C 180,E1 -15248.764,E2 -15248.764} C_VEL
LIN {X 0,Y 344.507,Z 266.271,A -85,B 0,C 180,E1 -15250.206,E2 -15250.206} C_VEL
LIN {X 0,Y 335.511,Z 249.065,A -85,B 0,C 180,E1 -15251.874,E2 -15251.874} C_VEL
LIN {X 0,Y 327.795,Z 235.626,A -85,B 0,C 180,E1 -15253.368,E2 -15253.368} C_VEL
LIN {X 0,Y 323.024,Z 227.494,A -85,B 0,C 180,E1 -15254.367,E2 -15254.367} C_VEL
LIN {X 0,Y 319.534,Z 217.988,A -85,B 0,C 180,E1 -15256.783,E2 -15256.783} C_VEL
LIN {X 0,Y 319.543,Z 217.986,A -85,B 0,C 180,E1 -15260.371,E2 -15260.371} C_VEL
LIN {X 0,Y 319.577,Z 217.976,A -85,B 0,C 180,E1 -15264.457,E2 -15264.457} C_VEL
LIN {X 0,Y 319.528,Z 217.975,A -85,B 0,C 180,E1 -15268.138,E2 -15268.138} C_VEL
LIN {X 0,Y 319.609,Z 217.986,A -85,B 0,C 180,E1 -15271.59,E2 -15271.59} C_VEL
LIN {X 0,Y 319.602,Z 217.969,A -85,B 0,C 180,E1 -15275.304,E2 -15275.304} C_VEL
LIN {X 0,Y 319.594,Z 217.987,A -85,B 0,C 180,E1 -15278.048,E2 -15278.048} C_VEL
LIN {X 0,Y 319.622,Z 217.963,A -85,B 0,C 180,E1 -15282.071,E2 -15282.071} C_VEL
LIN {X 0,Y 319.73,Z 217.958,A -85,B 0,C 180,E1 -15286.008,E2 -15286.008} C_VEL
LIN {X 0,Y 319.733,Z 217.945,A -85,B 0,C 180,E1 -15289.872,E2 -15289.872} C_VEL
LIN {X 0,Y 319.933,Z 217.942,A -85,B 0,C 180,E1 -15293.694,E2 -15293.694} C_VEL
LIN {X 0,Y 319.985,Z 217.893,A -85,B 0,C 180,E1 -15297.482,E2 -15297.482} C_VEL
LIN {X 0,Y 320.129,Z 217.91,A -85,B 0,C 180,E1 -15300,E2 -15300} C_VEL
LIN {X 0,Y 319.987,Z 217.935,A -85,B 0,C 180,E1 -15302.518,E2 -15302.518} C_VEL
LIN {X 0,Y 319.918,Z 217.931,A -85,B 0,C 180,E1 -15306.643,E2 -15306.643} C_VEL
LIN {X 0,Y 319.751,Z 217.957,A -85,B 0,C 180,E1 -15310.127,E2 -15310.127} C_VEL
LIN {X 0,Y 319.729,Z 217.968,A -85,B 0,C 180,E1 -15314.724,E2 -15314.724} C_VEL
LIN {X 0,Y 319.687,Z 217.95,A -85,B 0,C 180,E1 -15319.038,E2 -15319.038} C_VEL
LIN {X 0,Y 319.569,Z 217.987,A -85,B 0,C 180,E1 -15323.319,E2 -15323.319} C_VEL
LIN {X 0,Y 319.634,Z 217.962,A -85,B 0,C 180,E1 -15326.088,E2 -15326.088} C_VEL
LIN {X 0,Y 319.597,Z 217.986,A -85,B 0,C 180,E1 -15328.933,E2 -15328.933} C_VEL
LIN {X 0,Y 319.532,Z 217.975,A -85,B 0,C 180,E1 -15331.862,E2 -15331.862} C_VEL
LIN {X 0,Y 319.579,Z 217.991,A -85,B 0,C 180,E1 -15335.543,E2 -15335.543} C_VEL
LIN {X 0,Y 319.557,Z 217.983,A -85,B 0,C 180,E1 -15339.669,E2 -15339.669} C_VEL
LIN {X 0,Y 319.52,Z 217.981,A -85,B 0,C 180,E1 -15343.461,E2 -15343.461} C_VEL
LIN {X 0,Y 319.553,Z 217.994,A -85,B 0,C 180,E1 -15347.016,E2 -15347.016} C_VEL
LIN {X 0,Y 319.546,Z 217.99,A -85,B 0,C 180,E1 -15350.371,E2 -15350.371} C_VEL
LIN {X 0,Y 319.557,Z 217.976,A -85,B 0,C 180,E1 -15353.572,E2 -15353.572} C_VEL
LIN {X 0,Y 319.576,Z 217.991,A -85,B 0,C 180,E1 -15356.686,E2 -15356.686} C_VEL
LIN {X 0,Y 319.591,Z 217.98,A -85,B 0,C 180,E1 -15359.617,E2 -15359.617} C_VEL
LIN {X 0,Y 319.607,Z 217.975,A -85,B 0,C 180,E1 -15362.498,E2 -15362.498} C_VEL
LIN {X 0,Y 319.605,Z 217.982,A -85,B 0,C 180,E1 -15365.304,E2 -15365.304} C_VEL
LIN {X 0,Y 319.596,Z 217.989,A -85,B 0,C 180,E1 -15368.048,E2 -15368.048} C_VEL
LIN {X 0,Y 319.701,Z 217.938,A -85,B 0,C 180,E1 -15371.342,E2 -15371.342} C_VEL
LIN {X 0,Y 320.67,Z 220.766,A -85,B 0,C 180,E1 -15371.597,E2 -15371.597} C_VEL
LIN {X 0,Y 322.575,Z 223.21,A -85,B 0,C 180,E1 -15371.969,E2 -15371.969} C_VEL
LIN {X 0,Y 324.789,Z 226.618,A -85,B 0,C 180,E1 -15372.412,E2 -15372.412} C_VEL
LIN {X 0,Y 335.712,Z 243.613,A -85,B 0,C 180,E1 -15374.498,E2 -15374.498} C_VEL
LIN {X 0,Y 344.094,Z 257.902,A -85,B 0,C 180,E1 -15376.011,E2 -15376.011} C_VEL
LIN {X 0,Y 351.483,Z 272.548,A -85,B 0,C 180,E1 -15377.327,E2 -15377.327} C_VEL
LIN {X 0,Y 352.632,Z 275.039,A -85,B 0,C 180,E1 -15377.53,E2 -15377.53} C_VEL
LIN {X 0,Y 346.919,Z 419.059,A -85,B 0,C 180,E1 -15380.599,E2 -15380.599} C_VEL
LIN {X 0,Y 345.59,Z 436.18,A -85,B 0,C 180,E1 -15381.19,E2 -15381.19} C_VEL
LIN {X 0,Y 343.796,Z 452.702,A -85,B 0,C 180,E1 -15381.995,E2 -15381.995} C_VEL
LIN {X 0,Y 341.959,Z 467.125,A -85,B 0,C 180,E1 -15382.916,E2 -15382.916} C_VEL
LIN {X 0,Y 339.769,Z 481.693,A -85,B 0,C 180,E1 -15384.063,E2 -15384.063} C_VEL
LIN {X 0,Y 337.346,Z 495.28,A -85,B 0,C 180,E1 -15385.369,E2 -15385.369} C_VEL
LIN {X 0,Y 334.536,Z 509.319,A -85,B 0,C 180,E1 -15386.989,E2 -15386.989} C_VEL
LIN {X 0,Y 331.821,Z 522.248,A -85,B 0,C 180,E1 -15388.786,E2 -15388.786} C_VEL
LIN {X 0,Y 329.325,Z 533.412,A -85,B 0,C 180,E1 -15390.611,E2 -15390.611} C_VEL
LIN {X 0,Y 326.77,Z 544.49,A -85,B 0,C 180,E1 -15392.773,E2 -15392.773} C_VEL
LIN {X 0,Y 324.52,Z 554.112,A -85,B 0,C 180,E1 -15394.997,E2 -15394.997} C_VEL
LIN {X 0,Y 322.473,Z 563.236,A -85,B 0,C 180,E1 -15397.513,E2 -15397.513} C_VEL
LIN {X 0,Y 320.844,Z 570.985,A -85,B 0,C 180,E1 -15400.092,E2 -15400.092} C_VEL
LIN {X 0,Y 319.579,Z 577.323,A -85,B 0,C 180,E1 -15402.703,E2 -15402.703} C_VEL
LIN {X 0,Y 318.713,Z 582.471,A -85,B 0,C 180,E1 -15405.343,E2 -15405.343} C_VEL
LIN {X 0,Y 318.051,Z 586.702,A -85,B 0,C 180,E1 -15408.163,E2 -15408.163} C_VEL
LIN {X 0,Y 317.692,Z 589.379,A -85,B 0,C 180,E1 -15410.729,E2 -15410.729} C_VEL
LIN {X 0,Y 317.45,Z 591.185,A -85,B 0,C 180,E1 -15413.484,E2 -15413.484} C_VEL
LIN {X 0,Y 317.424,Z 591.881,A -85,B 0,C 180,E1 -15416.283,E2 -15416.283} C_VEL
LIN {X 0,Y 317.542,Z 591.335,A -85,B 0,C 180,E1 -15419.137,E2 -15419.137} C_VEL
LIN {X 0,Y 317.825,Z 589.573,A -85,B 0,C 180,E1 -15422.052,E2 -15422.052} C_VEL
LIN {X 0,Y 318.404,Z 586.479,A -85,B 0,C 180,E1 -15425.021,E2 -15425.021} C_VEL
LIN {X 0,Y 319.061,Z 582.736,A -85,B 0,C 180,E1 -15427.536,E2 -15427.536} C_VEL
LIN {X 0,Y 319.535,Z 580.381,A -85,B 0,C 180,E1 -15428.845,E2 -15428.845} C_VEL
LIN {X 0,Y 319.281,Z 578.513,A -85,B 0,C 180,E1 -15429.847,E2 -15429.847} C_VEL
LIN {X 0,Y 317.217,Z 575.309,A -85,B 0,C 180,E1 -15431.498,E2 -15431.498} C_VEL
LIN {X 0,Y 315.319,Z 571.757,A -85,B 0,C 180,E1 -15433.142,E2 -15433.142} C_VEL
LIN {X 0,Y 315.326,Z 569.216,A -85,B 0,C 180,E1 -15434.117,E2 -15434.117} C_VEL
LIN {X 0,Y 317.617,Z 560.611,A -85,B 0,C 180,E1 -15436.902,E2 -15436.902} C_VEL
LIN {X 0,Y 320.135,Z 551.654,A -85,B 0,C 180,E1 -15439.299,E2 -15439.299} C_VEL
LIN {X 0,Y 322.989,Z 541.506,A -85,B 0,C 180,E1 -15441.565,E2 -15441.565} C_VEL
LIN {X 0,Y 326.032,Z 530.235,A -85,B 0,C 180,E1 -15443.673,E2 -15443.673} C_VEL
LIN {X 0,Y 329.15,Z 518.248,A -85,B 0,C 180,E1 -15445.558,E2 -15445.558} C_VEL
LIN {X 0,Y 332.321,Z 505.179,A -85,B 0,C 180,E1 -15447.288,E2 -15447.288} C_VEL
LIN {X 0,Y 335.393,Z 491.267,A -85,B 0,C 180,E1 -15448.813,E2 -15448.813} C_VEL
LIN {X 0,Y 338.093,Z 477.284,A -85,B 0,C 180,E1 -15450.073,E2 -15450.073} C_VEL
LIN {X 0,Y 340.733,Z 461.378,A -85,B 0,C 180,E1 -15451.234,E2 -15451.234} C_VEL
LIN {X 0,Y 342.957,Z 444.774,A -85,B 0,C 180,E1 -15452.172,E2 -15452.172} C_VEL
LIN {X 0,Y 344.62,Z 429.05,A -85,B 0,C 180,E1 -15452.829,E2 -15452.829} C_VEL
LIN {X 0,Y 345.839,Z 411.806,A -85,B 0,C 180,E1 -15453.311,E2 -15453.311} C_VEL
LIN {X 0,Y 351.899,Z 280.374,A -85,B 0,C 180,E1 -15456.179,E2 -15456.179} C_VEL
LIN {X 0,Y 345.141,Z 267.078,A -85,B 0,C 180,E1 -15457.671,E2 -15457.671} C_VEL
LIN {X 0,Y 339.29,Z 256.863,A -85,B 0,C 180,E1 -15459.02,E2 -15459.02} C_VEL
LIN {X 0,Y 332.29,Z 246.212,A -85,B 0,C 180,E1 -15460.718,E2 -15460.718} C_VEL
LIN {X 0,Y 326.259,Z 237.745,A -85,B 0,C 180,E1 -15462.281,E2 -15462.281} C_VEL
LIN {X 0,Y 323.095,Z 233.466,A -85,B 0,C 180,E1 -15463.152,E2 -15463.152} C_VEL
LIN {X 0,Y 320.528,Z 229.967,A -85,B 0,C 180,E1 -15463.889,E2 -15463.889} C_VEL
LIN {X 0,Y 319.698,Z 228.894,A -85,B 0,C 180,E1 -15464.132,E2 -15464.132} C_VEL
LIN {X 0,Y 317.347,Z 226.103,A -85,B 0,C 180,E1 -15464.828,E2 -15464.828} C_VEL
LIN {X 0,Y 316.275,Z 224.169,A -85,B 0,C 180,E1 -15465.18,E2 -15465.18} C_VEL
LIN {X 0,Y 313.982,Z 222.141,A -85,B 0,C 180,E1 -15465.87,E2 -15465.87} C_VEL
LIN {X 0,Y 312.864,Z 219.834,A -85,B 0,C 180,E1 -15466.275,E2 -15466.275} C_VEL
LIN {X 0,Y 312.666,Z 218.849,A -85,B 0,C 180,E1 -15466.431,E2 -15466.431} C_VEL
LIN {X 0,Y 312.745,Z 218.838,A -85,B 0,C 180,E1 -15470.95,E2 -15470.95} C_VEL
LIN {X 0,Y 312.885,Z 218.819,A -85,B 0,C 180,E1 -15473.552,E2 -15473.552} C_VEL
LIN {X 0,Y 312.929,Z 218.816,A -85,B 0,C 180,E1 -15477.426,E2 -15477.426} C_VEL
LIN {X 0,Y 313.096,Z 218.794,A -85,B 0,C 180,E1 -15480,E2 -15480} C_VEL
LIN {X 0,Y 312.93,Z 218.814,A -85,B 0,C 180,E1 -15482.574,E2 -15482.574} C_VEL
LIN {X 0,Y 312.895,Z 218.82,A -85,B 0,C 180,E1 -15486.448,E2 -15486.448} C_VEL
LIN {X 0,Y 312.762,Z 218.836,A -85,B 0,C 180,E1 -15489.05,E2 -15489.05} C_VEL
LIN {X 0,Y 312.629,Z 218.854,A -85,B 0,C 180,E1 -15492.991,E2 -15492.991} C_VEL
LIN {X 0,Y 312.633,Z 218.853,A -85,B 0,C 180,E1 -15495.65,E2 -15495.65} C_VEL
LIN {X 0,Y 312.625,Z 218.85,A -85,B 0,C 180,E1 -15499.236,E2 -15499.236} C_VEL
LIN {X 0,Y 312.541,Z 218.867,A -85,B 0,C 180,E1 -15502.789,E2 -15502.789} C_VEL
LIN {X 0,Y 312.597,Z 218.858,A -85,B 0,C 180,E1 -15505.936,E2 -15505.936} C_VEL
LIN {X 0,Y 312.533,Z 218.866,A -85,B 0,C 180,E1 -15509.651,E2 -15509.651} C_VEL
LIN {X 0,Y 312.515,Z 218.869,A -85,B 0,C 180,E1 -15513.689,E2 -15513.689} C_VEL
LIN {X 0,Y 312.515,Z 218.875,A -85,B 0,C 180,E1 -15517.386,E2 -15517.386} C_VEL
LIN {X 0,Y 312.526,Z 219.022,A -85,B 0,C 180,E1 -15517.867,E2 -15517.867} C_VEL
LIN {X 0,Y 315.326,Z 225.522,A -85,B 0,C 180,E1 -15520.267,E2 -15520.267} C_VEL
LIN {X 0,Y 320.213,Z 232.334,A -85,B 0,C 180,E1 -15521.765,E2 -15521.765} C_VEL
LIN {X 0,Y 325.502,Z 240.136,A -85,B 0,C 180,E1 -15523.277,E2 -15523.277} C_VEL
LIN {X 0,Y 332.141,Z 250.404,A -85,B 0,C 180,E1 -15525.034,E2 -15525.034} C_VEL
LIN {X 0,Y 339.187,Z 262.428,A -85,B 0,C 180,E1 -15526.778,E2 -15526.778} C_VEL
LIN {X 0,Y 346.738,Z 276.937,A -85,B 0,C 180,E1 -15528.534,E2 -15528.534} C_VEL
LIN {X 0,Y 351.674,Z 287.548,A -85,B 0,C 180,E1 -15529.632,E2 -15529.632} C_VEL
LIN {X 0,Y 346.853,Z 390.872,A -85,B 0,C 180,E1 -15531.877,E2 -15531.877} C_VEL
LIN {X 0,Y 344.784,Z 435.803,A -85,B 0,C 180,E1 -15532.899,E2 -15532.899} C_VEL
LIN {X 0,Y 342.997,Z 453.29,A -85,B 0,C 180,E1 -15533.487,E2 -15533.487} C_VEL
LIN {X 0,Y 340.832,Z 469.553,A -85,B 0,C 180,E1 -15534.282,E2 -15534.282} C_VEL
LIN {X 0,Y 338.555,Z 483.822,A -85,B 0,C 180,E1 -15535.19,E2 -15535.19} C_VEL
LIN {X 0,Y 335.788,Z 498.294,A -85,B 0,C 180,E1 -15536.315,E2 -15536.315} C_VEL
LIN {X 0,Y 332.753,Z 512.622,A -85,B 0,C 180,E1 -15537.699,E2 -15537.699} C_VEL
LIN {X 0,Y 329.394,Z 526.895,A -85,B 0,C 180,E1 -15539.377,E2 -15539.377} C_VEL
LIN {X 0,Y 326.446,Z 538.664,A -85,B 0,C 180,E1 -15541.028,E2 -15541.028} C_VEL
LIN {X 0,Y 323.275,Z 550.815,A -85,B 0,C 180,E1 -15543.042,E2 -15543.042} C_VEL
LIN {X 0,Y 320.189,Z 562.408,A -85,B 0,C 180,E1 -15545.353,E2 -15545.353} C_VEL
LIN {X 0,Y 317.365,Z 572.951,A -85,B 0,C 180,E1 -15547.886,E2 -15547.886} C_VEL
LIN {X 0,Y 315.192,Z 581.832,A -85,B 0,C 180,E1 -15550.461,E2 -15550.461} C_VEL
LIN {X 0,Y 313.421,Z 589.305,A -85,B 0,C 180,E1 -15553.053,E2 -15553.053} C_VEL
LIN {X 0,Y 312.183,Z 595.471,A -85,B 0,C 180,E1 -15555.663,E2 -15555.663} C_VEL
LIN {X 0,Y 311.378,Z 600.435,A -85,B 0,C 180,E1 -15558.28,E2 -15558.28} C_VEL
LIN {X 0,Y 310.873,Z 604.372,A -85,B 0,C 180,E1 -15560.895,E2 -15560.895} C_VEL
LIN {X 0,Y 310.722,Z 607.958,A -85,B 0,C 180,E1 -15564.385,E2 -15564.385} C_VEL
LIN {X 0,Y 310.674,Z 609.588,A -85,B 0,C 180,E1 -15567.407,E2 -15567.407} C_VEL
LIN {X 0,Y 310.69,Z 609.959,A -85,B 0,C 180,E1 -15570,E2 -15570} C_VEL
LIN {X 0,Y 310.677,Z 609.342,A -85,B 0,C 180,E1 -15572.593,E2 -15572.593} C_VEL
LIN {X 0,Y 310.722,Z 607.36,A -85,B 0,C 180,E1 -15575.616,E2 -15575.616} C_VEL
LIN {X 0,Y 310.772,Z 605.108,A -85,B 0,C 180,E1 -15577.799,E2 -15577.799} C_VEL
LIN {X 0,Y 311.18,Z 600.323,A -85,B 0,C 180,E1 -15581.068,E2 -15581.068} C_VEL
LIN {X 0,Y 311.955,Z 595.227,A -85,B 0,C 180,E1 -15583.683,E2 -15583.683} C_VEL
LIN {X 0,Y 312.975,Z 588.956,A -85,B 0,C 180,E1 -15586.302,E2 -15586.302} C_VEL
LIN {X 0,Y 314.777,Z 580.225,A -85,B 0,C 180,E1 -15589.228,E2 -15589.228} C_VEL
LIN {X 0,Y 316.79,Z 570.789,A -85,B 0,C 180,E1 -15591.814,E2 -15591.814} C_VEL
LIN {X 0,Y 319.066,Z 561.062,A -85,B 0,C 180,E1 -15594.048,E2 -15594.048} C_VEL
LIN {X 0,Y 321.631,Z 550.401,A -85,B 0,C 180,E1 -15596.129,E2 -15596.129} C_VEL
LIN {X 0,Y 323.887,Z 540.308,A -85,B 0,C 180,E1 -15597.809,E2 -15597.809} C_VEL
LIN {X 0,Y 326.815,Z 527.352,A -85,B 0,C 180,E1 -15599.644,E2 -15599.644} C_VEL
LIN {X 0,Y 329.743,Z 513.615,A -85,B 0,C 180,E1 -15601.265,E2 -15601.265} C_VEL
LIN {X 0,Y 332.739,Z 498.041,A -85,B 0,C 180,E1 -15602.768,E2 -15602.768} C_VEL
LIN {X 0,Y 335.394,Z 482.043,A -85,B 0,C 180,E1 -15604.002,E2 -15604.002} C_VEL
LIN {X 0,Y 337.498,Z 466.626,A -85,B 0,C 180,E1 -15604.935,E2 -15604.935} C_VEL
LIN {X 0,Y 339.272,Z 451.3,A -85,B 0,C 180,E1 -15605.638,E2 -15605.638} C_VEL
LIN {X 0,Y 340.669,Z 436.058,A -85,B 0,C 180,E1 -15606.141,E2 -15606.141} C_VEL
LIN {X 0,Y 346.771,Z 285.484,A -85,B 0,C 180,E1 -15609.405,E2 -15609.405} C_VEL
LIN {X 0,Y 339.35,Z 269.847,A -85,B 0,C 180,E1 -15610.774,E2 -15610.774} C_VEL
LIN {X 0,Y 330.649,Z 253.099,A -85,B 0,C 180,E1 -15612.443,E2 -15612.443} C_VEL
LIN {X 0,Y 321.27,Z 236.666,A -85,B 0,C 180,E1 -15614.326,E2 -15614.326} C_VEL
LIN {X 0,Y 315.556,Z 227.235,A -85,B 0,C 180,E1 -15615.562,E2 -15615.562} C_VEL
LIN {X 0,Y 312.478,Z 218.875,A -85,B 0,C 180,E1 -15617.798,E2 -15617.798} C_VEL
LIN {X 0,Y 312.493,Z 218.872,A -85,B 0,C 180,E1 -15620.971,E2 -15620.971} C_VEL
LIN {X 0,Y 312.529,Z 218.851,A -85,B 0,C 180,E1 -15624.22,E2 -15624.22} C_VEL
LIN {X 0,Y 312.502,Z 218.856,A -85,B 0,C 180,E1 -15627.334,E2 -15627.334} C_VEL
LIN {X 0,Y 312.543,Z 218.867,A -85,B 0,C 180,E1 -15631.279,E2 -15631.279} C_VEL
LIN {X 0,Y 312.583,Z 218.836,A -85,B 0,C 180,E1 -15634.711,E2 -15634.711} C_VEL
LIN {X 0,Y 312.586,Z 218.861,A -85,B 0,C 180,E1 -15637.529,E2 -15637.529} C_VEL
LIN {X 0,Y 312.58,Z 218.834,A -85,B 0,C 180,E1 -15641.653,E2 -15641.653} C_VEL
LIN {X 0,Y 312.683,Z 218.841,A -85,B 0,C 180,E1 -15645.686,E2 -15645.686} C_VEL
LIN {X 0,Y 312.683,Z 218.818,A -85,B 0,C 180,E1 -15649.641,E2 -15649.641} C_VEL
LIN {X 0,Y 312.889,Z 218.82,A -85,B 0,C 180,E1 -15653.552,E2 -15653.552} C_VEL
LIN {X 0,Y 312.932,Z 218.77,A -85,B 0,C 180,E1 -15657.426,E2 -15657.426} C_VEL
LIN {X 0,Y 313.082,Z 218.788,A -85,B 0,C 180,E1 -15660,E2 -15660} C_VEL
LIN {X 0,Y 312.933,Z 218.813,A -85,B 0,C 180,E1 -15662.574,E2 -15662.574} C_VEL
LIN {X 0,Y 312.883,Z 218.807,A -85,B 0,C 180,E1 -15666.624,E2 -15666.624} C_VEL
LIN {X 0,Y 312.766,Z 218.835,A -85,B 0,C 180,E1 -15669.05,E2 -15669.05} C_VEL
LIN {X 0,Y 312.632,Z 218.836,A -85,B 0,C 180,E1 -15672.991,E2 -15672.991} C_VEL
LIN {X 0,Y 312.637,Z 218.853,A -85,B 0,C 180,E1 -15675.65,E2 -15675.65} C_VEL
LIN {X 0,Y 312.628,Z 218.83,A -85,B 0,C 180,E1 -15679.236,E2 -15679.236} C_VEL
LIN {X 0,Y 312.544,Z 218.863,A -85,B 0,C 180,E1 -15682.789,E2 -15682.789} C_VEL
LIN {X 0,Y 312.585,Z 218.846,A -85,B 0,C 180,E1 -15686.722,E2 -15686.722} C_VEL
LIN {X 0,Y 312.547,Z 218.863,A -85,B 0,C 180,E1 -15689.65,E2 -15689.65} C_VEL
LIN {X 0,Y 312.518,Z 218.859,A -85,B 0,C 180,E1 -15693.689,E2 -15693.689} C_VEL
LIN {X 0,Y 312.519,Z 218.852,A -85,B 0,C 180,E1 -15697.386,E2 -15697.386} C_VEL
LIN {X 0,Y 312.489,Z 218.872,A -85,B 0,C 180,E1 -15700.709,E2 -15700.709} C_VEL
LIN {X 0,Y 312.45,Z 218.861,A -85,B 0,C 180,E1 -15704.21,E2 -15704.21} C_VEL
LIN {X 0,Y 312.483,Z 218.864,A -85,B 0,C 180,E1 -15707.919,E2 -15707.919} C_VEL
LIN {X 0,Y 312.504,Z 218.869,A -85,B 0,C 180,E1 -15711.917,E2 -15711.917} C_VEL
LIN {X 0,Y 312.531,Z 218.851,A -85,B 0,C 180,E1 -15714.22,E2 -15714.22} C_VEL
LIN {X 0,Y 312.503,Z 218.865,A -85,B 0,C 180,E1 -15717.334,E2 -15717.334} C_VEL
LIN {X 0,Y 312.551,Z 218.864,A -85,B 0,C 180,E1 -15721.276,E2 -15721.276} C_VEL
LIN {X 0,Y 312.585,Z 218.862,A -85,B 0,C 180,E1 -15724.711,E2 -15724.711} C_VEL
LIN {X 0,Y 312.587,Z 218.858,A -85,B 0,C 180,E1 -15727.529,E2 -15727.529} C_VEL
